KUKA KRL program: EPS_2_25694_BR02_A_20251117072400.src

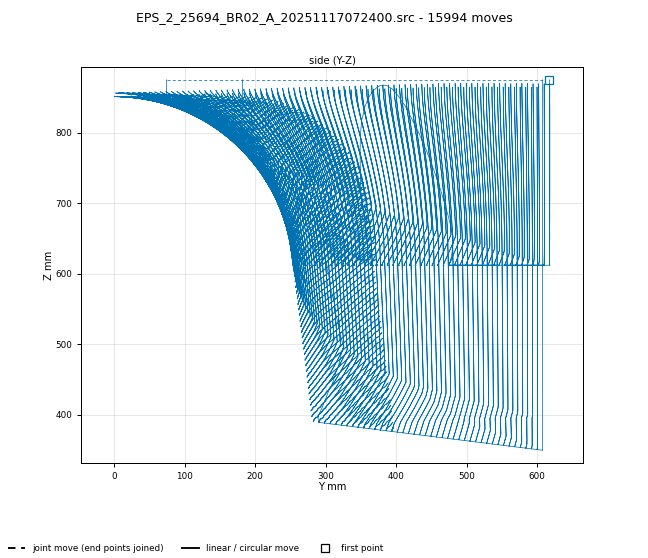
[picture p0: tool path of EPS_2_25694_BR02_A_20251117072400.src, 15994 of 15996 moves have a stored position in this frame; points joined in program order, loops and branches not executed]
&ACCESS RVP
&REL 4
&COMMENT QRS 19112012
&PARAM EDITMASK = *
DEF PART()
EXT BAS (BAS_COMMAND :IN,REAL :IN )
INT I
BAS (#INITMOV,0 )

;KUKA QRS Post kuka4.cps  Date:22-06-2017 !

File_ID=2912

QRS_PRE_INIT()

;Init var - Until changes are made in qrs_pre_init
Outlet_Square_prg=0
Inlet_1_Square_prg=0
Inlet_2_Square_prg=0
Inlet_3_Square_prg=0
Inlet_4_Square_prg=0
Inlet_5_Square_prg=0

Outlet_1={X 0.000, Y 466.000, Z 636.500, B 0.000, E1 0.000 }
Inlet_1={X 0.000, Y 492.670, Z 611.500, B 0.000, E1 180.000 }
Outlet_1_type=457
Inlet_1_type=0
;QRS#1=Sidecore dimensions
;QRS#2=450-18" Concrete
;QRS#3=DeadEnd 457
;QRS#4=
;QRS#5=
;QRS#6=
;QRS#7=
;QRS#8=
;QRS#9=28A PSX-2
;QRS#10=

;QRS#11=
;QRS#12=
;QRS#13=
;QRS#14=
;QRS#15=
;QRS#16=1220x127x1219 4'
;QRS#17=EPS Height
;QRS#18=865
;QRS#19=*
;QRS#20= UPDATED VERSION 22-06-2017
;QRS#21=*
Outlet_Square=0250
Inlet_1_Square=00
Inlet_2_Square=0
Inlet_3_Square=0
Inlet_4_Square=0
Inlet_5_Square=0
Mill_Square=1
Outlet_Square_Prg=274
Inlet_1_Square_prg=0

QRS_INIT()

$ADVANCE=5

; T1
PTP {E1 171.224,E2 171.224}
PTP {X 0,Y 617.539,A -85,B 0,C 180,E1 171.224,E2 171.224,E3 0,E4 0,E5 0,E6 0}
QRS_SPEED_INIT()
LIN {X 0,Y 617.539,Z 875,A -85,B 0,C 180,E1 171.224,E2 171.224,E3 0,E4 0,E5 0,E6 0} C_VEL
LIN {X 0,Y 617.539,Z 613.91,A -85,B 0,C 180,E1 171.224,E2 171.224} C_VEL
LIN {X 0,Y 617.52,Z 611.91,A -85,B 0,C 180,E1 171.41,E2 171.41} C_VEL
LIN {X 0,Y 618.01,Z 611.91,A -85,B 0,C 180,E1 174.219,E2 174.219} C_VEL
LIN {X 0,Y 618.036,Z 611.91,A -85,B 0,C 180,E1 178.849,E2 178.849} C_VEL
LIN {X 0,Y 617.996,Z 611.91,A -85,B 0,C 180,E1 183.472,E2 183.472} C_VEL
LIN {X 0,Y 617.993,Z 611.91,A -85,B 0,C 180,E1 188.118,E2 188.118} C_VEL
LIN {X 0,Y 617.979,Z 611.91,A -85,B 0,C 180,E1 192.819,E2 192.819} C_VEL
LIN {X 0,Y 617.92,Z 611.91,A -85,B 0,C 180,E1 197.611,E2 197.611} C_VEL
LIN {X 0,Y 617.739,Z 611.91,A -85,B 0,C 180,E1 198.543,E2 198.543} C_VEL
LIN {X 0,Y 617.926,Z 611.91,A -85,B 0,C 180,E1 202.533,E2 202.533} C_VEL
LIN {X 0,Y 617.417,Z 611.91,A -85,B 0,C 180,E1 205.081,E2 205.081} C_VEL
LIN {X 0,Y 617.847,Z 611.91,A -85,B 0,C 180,E1 207.641,E2 207.641} C_VEL
LIN {X 0,Y 617.342,Z 611.91,A -85,B 0,C 180,E1 210.31,E2 210.31} C_VEL
LIN {X 0,Y 617.812,Z 611.91,A -85,B 0,C 180,E1 213,E2 213} C_VEL
LIN {X 0,Y 617.679,Z 611.91,A -85,B 0,C 180,E1 214.194,E2 214.194} C_VEL
LIN {X 0,Y 617.782,Z 611.91,A -85,B 0,C 180,E1 218.707,E2 218.707} C_VEL
LIN {X 0,Y 617.421,Z 611.91,A -85,B 0,C 180,E1 221.764,E2 221.764} C_VEL
LIN {X 0,Y 617.823,Z 611.91,A -85,B 0,C 180,E1 224.908,E2 224.908} C_VEL
LIN {X 0,Y 617.772,Z 611.91,A -85,B 0,C 180,E1 228.277,E2 228.277} C_VEL
LIN {X 0,Y 617.551,Z 611.91,A -85,B 0,C 180,E1 231.279,E2 231.279} C_VEL
LIN {X 0,Y 617.574,Z 611.91,A -85,B 0,C 180,E1 231.903,E2 231.903} C_VEL
LIN {X 0,Y 617.811,Z 611.91,A -85,B 0,C 180,E1 234.203,E2 234.203} C_VEL
LIN {X 0,Y 617.347,Z 611.91,A -85,B 0,C 180,E1 236.976,E2 236.976} C_VEL
LIN {X 0,Y 617.893,Z 611.91,A -85,B 0,C 180,E1 239.723,E2 239.723} C_VEL
LIN {X 0,Y 618.039,Z 611.91,A -85,B 0,C 180,E1 244.95,E2 244.95} C_VEL
LIN {X 0,Y 617.661,Z 611.91,A -85,B 0,C 180,E1 245.064,E2 245.064} C_VEL
LIN {X 0,Y 617.895,Z 648.089,A -85,B 0,C 180,E1 245.541,E2 245.541} C_VEL
LIN {X 0,Y 617.86,Z 657.573,A -85,B 0,C 180,E1 245.694,E2 245.694} C_VEL
LIN {X 0,Y 617.789,Z 666.269,A -85,B 0,C 180,E1 245.863,E2 245.863} C_VEL
LIN {X 0,Y 617.896,Z 680.361,A -85,B 0,C 180,E1 246.223,E2 246.223} C_VEL
LIN {X 0,Y 617.817,Z 691.301,A -85,B 0,C 180,E1 246.552,E2 246.552} C_VEL
LIN {X 0,Y 617.928,Z 701.625,A -85,B 0,C 180,E1 246.918,E2 246.918} C_VEL
LIN {X 0,Y 617.942,Z 713.385,A -85,B 0,C 180,E1 247.393,E2 247.393} C_VEL
LIN {X 0,Y 617.876,Z 723.675,A -85,B 0,C 180,E1 247.859,E2 247.859} C_VEL
LIN {X 0,Y 617.946,Z 734.343,A -85,B 0,C 180,E1 248.407,E2 248.407} C_VEL
LIN {X 0,Y 617.967,Z 745.217,A -85,B 0,C 180,E1 249.027,E2 249.027} C_VEL
LIN {X 0,Y 617.938,Z 755.026,A -85,B 0,C 180,E1 249.644,E2 249.644} C_VEL
LIN {X 0,Y 617.951,Z 764.54,A -85,B 0,C 180,E1 250.302,E2 250.302} C_VEL
LIN {X 0,Y 617.956,Z 773.748,A -85,B 0,C 180,E1 251.001,E2 251.001} C_VEL
LIN {X 0,Y 617.967,Z 782.099,A -85,B 0,C 180,E1 251.691,E2 251.691} C_VEL
LIN {X 0,Y 617.941,Z 791.033,A -85,B 0,C 180,E1 252.497,E2 252.497} C_VEL
LIN {X 0,Y 617.896,Z 798.436,A -85,B 0,C 180,E1 253.222,E2 253.222} C_VEL
LIN {X 0,Y 617.951,Z 806.146,A -85,B 0,C 180,E1 254.049,E2 254.049} C_VEL
LIN {X 0,Y 617.974,Z 812.663,A -85,B 0,C 180,E1 254.803,E2 254.803} C_VEL
LIN {X 0,Y 617.884,Z 819.776,A -85,B 0,C 180,E1 255.697,E2 255.697} C_VEL
LIN {X 0,Y 617.866,Z 826.241,A -85,B 0,C 180,E1 256.589,E2 256.589} C_VEL
LIN {X 0,Y 617.965,Z 832.102,A -85,B 0,C 180,E1 257.481,E2 257.481} C_VEL
LIN {X 0,Y 617.877,Z 837.463,A -85,B 0,C 180,E1 258.365,E2 258.365} C_VEL
LIN {X 0,Y 617.831,Z 843.766,A -85,B 0,C 180,E1 259.542,E2 259.542} C_VEL
LIN {X 0,Y 617.913,Z 847.34,A -85,B 0,C 180,E1 260.283,E2 260.283} C_VEL
LIN {X 0,Y 617.929,Z 852.374,A -85,B 0,C 180,E1 261.453,E2 261.453} C_VEL
LIN {X 0,Y 617.831,Z 855.756,A -85,B 0,C 180,E1 262.35,E2 262.35} C_VEL
LIN {X 0,Y 617.936,Z 860.15,A -85,B 0,C 180,E1 263.748,E2 263.748} C_VEL
LIN {X 0,Y 617.913,Z 862.617,A -85,B 0,C 180,E1 264.677,E2 264.677} C_VEL
LIN {X 0,Y 617.775,Z 865.488,A -85,B 0,C 180,E1 266.068,E2 266.068} C_VEL
LIN {X 0,Y 617.811,Z 866.258,A -85,B 0,C 180,E1 266.531,E2 266.531} C_VEL
LIN {X 0,Y 617.948,Z 867.966,A -85,B 0,C 180,E1 267.92,E2 267.92} C_VEL
LIN {X 0,Y 617.798,Z 868.661,A -85,B 0,C 180,E1 268.844,E2 268.844} C_VEL
LIN {X 0,Y 617.834,Z 868.908,A -85,B 0,C 180,E1 270.231,E2 270.231} C_VEL
LIN {X 0,Y 617.983,Z 868.61,A -85,B 0,C 180,E1 271.155,E2 271.155} C_VEL
LIN {X 0,Y 617.813,Z 867.476,A -85,B 0,C 180,E1 272.543,E2 272.543} C_VEL
LIN {X 0,Y 617.843,Z 866.25,A -85,B 0,C 180,E1 273.469,E2 273.469} C_VEL
LIN {X 0,Y 617.982,Z 864.618,A -85,B 0,C 180,E1 274.395,E2 274.395} C_VEL
LIN {X 0,Y 617.84,Z 862.636,A -85,B 0,C 180,E1 275.323,E2 275.323} C_VEL
LIN {X 0,Y 617.779,Z 860.19,A -85,B 0,C 180,E1 276.253,E2 276.253} C_VEL
LIN {X 0,Y 617.946,Z 855.728,A -85,B 0,C 180,E1 277.648,E2 277.648} C_VEL
LIN {X 0,Y 617.875,Z 851.36,A -85,B 0,C 180,E1 278.793,E2 278.793} C_VEL
LIN {X 0,Y 617.822,Z 847.625,A -85,B 0,C 180,E1 279.664,E2 279.664} C_VEL
LIN {X 0,Y 617.935,Z 842.258,A -85,B 0,C 180,E1 280.75,E2 280.75} C_VEL
LIN {X 0,Y 617.942,Z 837.449,A -85,B 0,C 180,E1 281.634,E2 281.634} C_VEL
LIN {X 0,Y 617.865,Z 830.198,A -85,B 0,C 180,E1 282.818,E2 282.818} C_VEL
LIN {X 0,Y 617.941,Z 824.137,A -85,B 0,C 180,E1 283.706,E2 283.706} C_VEL
LIN {X 0,Y 617.959,Z 817.47,A -85,B 0,C 180,E1 284.6,E2 284.6} C_VEL
LIN {X 0,Y 617.884,Z 809.516,A -85,B 0,C 180,E1 285.57,E2 285.57} C_VEL
LIN {X 0,Y 617.919,Z 802.465,A -85,B 0,C 180,E1 286.355,E2 286.355} C_VEL
LIN {X 0,Y 617.972,Z 794.297,A -85,B 0,C 180,E1 287.187,E2 287.187} C_VEL
LIN {X 0,Y 617.934,Z 787.157,A -85,B 0,C 180,E1 287.863,E2 287.863} C_VEL
LIN {X 0,Y 617.923,Z 778.285,A -85,B 0,C 180,E1 288.631,E2 288.631} C_VEL
LIN {X 0,Y 617.943,Z 769.373,A -85,B 0,C 180,E1 289.338,E2 289.338} C_VEL
LIN {X 0,Y 617.96,Z 760.865,A -85,B 0,C 180,E1 289.959,E2 289.959} C_VEL
LIN {X 0,Y 617.96,Z 751.47,A -85,B 0,C 180,E1 290.587,E2 290.587} C_VEL
LIN {X 0,Y 617.918,Z 741.279,A -85,B 0,C 180,E1 291.207,E2 291.207} C_VEL
LIN {X 0,Y 617.943,Z 731.417,A -85,B 0,C 180,E1 291.749,E2 291.749} C_VEL
LIN {X 0,Y 617.958,Z 720.361,A -85,B 0,C 180,E1 292.294,E2 292.294} C_VEL
LIN {X 0,Y 617.921,Z 709.648,A -85,B 0,C 180,E1 292.766,E2 292.766} C_VEL
LIN {X 0,Y 617.818,Z 698.36,A -85,B 0,C 180,E1 293.205,E2 293.205} C_VEL
LIN {X 0,Y 617.93,Z 686.204,A -85,B 0,C 180,E1 293.604,E2 293.604} C_VEL
LIN {X 0,Y 617.911,Z 675,A -85,B 0,C 180,E1 293.92,E2 293.92} C_VEL
LIN {X 0,Y 617.75,Z 663.936,A -85,B 0,C 180,E1 294.186,E2 294.186} C_VEL
LIN {X 0,Y 617.899,Z 651.747,A -85,B 0,C 180,E1 294.405,E2 294.405} C_VEL
LIN {X 0,Y 617.853,Z 635.322,A -85,B 0,C 180,E1 294.632,E2 294.632} C_VEL
LIN {X 0,Y 617.679,Z 611.91,A -85,B 0,C 180,E1 294.936,E2 294.936} C_VEL
LIN {X 0,Y 618.055,Z 611.91,A -85,B 0,C 180,E1 295.049,E2 295.049} C_VEL
LIN {X 0,Y 617.893,Z 611.91,A -85,B 0,C 180,E1 300.277,E2 300.277} C_VEL
LIN {X 0,Y 617.347,Z 611.91,A -85,B 0,C 180,E1 303.024,E2 303.024} C_VEL
LIN {X 0,Y 617.811,Z 611.91,A -85,B 0,C 180,E1 305.797,E2 305.797} C_VEL
LIN {X 0,Y 617.546,Z 611.91,A -85,B 0,C 180,E1 308.721,E2 308.721} C_VEL
LIN {X 0,Y 617.75,Z 611.91,A -85,B 0,C 180,E1 311.733,E2 311.733} C_VEL
LIN {X 0,Y 617.804,Z 611.91,A -85,B 0,C 180,E1 315.09,E2 315.09} C_VEL
LIN {X 0,Y 617.418,Z 611.91,A -85,B 0,C 180,E1 318.31,E2 318.31} C_VEL
LIN {X 0,Y 617.776,Z 611.91,A -85,B 0,C 180,E1 321.292,E2 321.292} C_VEL
LIN {X 0,Y 617.679,Z 611.91,A -85,B 0,C 180,E1 325.806,E2 325.806} C_VEL
LIN {X 0,Y 617.847,Z 611.91,A -85,B 0,C 180,E1 327.002,E2 327.002} C_VEL
LIN {X 0,Y 617.633,Z 611.91,A -85,B 0,C 180,E1 330.175,E2 330.175} C_VEL
LIN {X 0,Y 617.65,Z 611.91,A -85,B 0,C 180,E1 332.349,E2 332.349} C_VEL
LIN {X 0,Y 617.509,Z 611.91,A -85,B 0,C 180,E1 335.241,E2 335.241} C_VEL
LIN {X 0,Y 617.715,Z 611.91,A -85,B 0,C 180,E1 337.459,E2 337.459} C_VEL
LIN {X 0,Y 617.711,Z 611.91,A -85,B 0,C 180,E1 341.465,E2 341.465} C_VEL
LIN {X 0,Y 617.915,Z 611.91,A -85,B 0,C 180,E1 342.389,E2 342.389} C_VEL
LIN {X 0,Y 617.972,Z 611.91,A -85,B 0,C 180,E1 347.181,E2 347.181} C_VEL
LIN {X 0,Y 617.987,Z 611.91,A -85,B 0,C 180,E1 351.882,E2 351.882} C_VEL
LIN {X 0,Y 617.986,Z 611.91,A -85,B 0,C 180,E1 356.528,E2 356.528} C_VEL
LIN {X 0,Y 618.036,Z 611.91,A -85,B 0,C 180,E1 361.151,E2 361.151} C_VEL
LIN {X 0,Y 618.009,Z 611.91,A -85,B 0,C 180,E1 365.781,E2 365.781} C_VEL
LIN {X 0,Y 617.945,Z 611.91,A -85,B 0,C 180,E1 370.451,E2 370.451} C_VEL
LIN {X 0,Y 617.949,Z 611.91,A -85,B 0,C 180,E1 375.192,E2 375.192} C_VEL
LIN {X 0,Y 617.917,Z 611.91,A -85,B 0,C 180,E1 380.044,E2 380.044} C_VEL
LIN {X 0,Y 617.427,Z 611.91,A -85,B 0,C 180,E1 382.542,E2 382.542} C_VEL
LIN {X 0,Y 617.87,Z 611.91,A -85,B 0,C 180,E1 385.051,E2 385.051} C_VEL
LIN {X 0,Y 617.368,Z 611.91,A -85,B 0,C 180,E1 387.654,E2 387.654} C_VEL
LIN {X 0,Y 617.822,Z 611.91,A -85,B 0,C 180,E1 390.274,E2 390.274} C_VEL
LIN {X 0,Y 617.306,Z 611.91,A -85,B 0,C 180,E1 393.02,E2 393.02} C_VEL
LIN {X 0,Y 617.795,Z 611.91,A -85,B 0,C 180,E1 395.791,E2 395.791} C_VEL
LIN {X 0,Y 617.874,Z 611.91,A -85,B 0,C 180,E1 398.689,E2 398.689} C_VEL
LIN {X 0,Y 617.401,Z 611.91,A -85,B 0,C 180,E1 401.754,E2 401.754} C_VEL
LIN {X 0,Y 617.853,Z 611.91,A -85,B 0,C 180,E1 404.893,E2 404.893} C_VEL
LIN {X 0,Y 617.725,Z 611.91,A -85,B 0,C 180,E1 408.269,E2 408.269} C_VEL
LIN {X 0,Y 617.496,Z 611.91,A -85,B 0,C 180,E1 411.275,E2 411.275} C_VEL
LIN {X 0,Y 617.519,Z 611.91,A -85,B 0,C 180,E1 411.895,E2 411.895} C_VEL
LIN {X 0,Y 617.754,Z 611.91,A -85,B 0,C 180,E1 414.199,E2 414.199} C_VEL
LIN {X 0,Y 617.28,Z 611.91,A -85,B 0,C 180,E1 416.972,E2 416.972} C_VEL
LIN {X 0,Y 617.815,Z 611.91,A -85,B 0,C 180,E1 419.719,E2 419.719} C_VEL
LIN {X 0,Y 617.39,Z 611.91,A -85,B 0,C 180,E1 422.34,E2 422.34} C_VEL
LIN {X 0,Y 617.915,Z 611.91,A -85,B 0,C 180,E1 424.945,E2 424.945} C_VEL
LIN {X 0,Y 617.43,Z 611.91,A -85,B 0,C 180,E1 427.452,E2 427.452} C_VEL
LIN {X 0,Y 617.885,Z 611.91,A -85,B 0,C 180,E1 429.95,E2 429.95} C_VEL
LIN {X 0,Y 617.964,Z 611.91,A -85,B 0,C 180,E1 434.803,E2 434.803} C_VEL
LIN {X 0,Y 617.954,Z 611.91,A -85,B 0,C 180,E1 439.544,E2 439.544} C_VEL
LIN {X 0,Y 617.973,Z 611.91,A -85,B 0,C 180,E1 444.213,E2 444.213} C_VEL
LIN {X 0,Y 618.038,Z 611.91,A -85,B 0,C 180,E1 448.845,E2 448.845} C_VEL
LIN {X 0,Y 618.005,Z 611.91,A -85,B 0,C 180,E1 453.468,E2 453.468} C_VEL
LIN {X 0,Y 617.96,Z 611.91,A -85,B 0,C 180,E1 458.115,E2 458.115} C_VEL
LIN {X 0,Y 617.98,Z 611.91,A -85,B 0,C 180,E1 462.815,E2 462.815} C_VEL
LIN {X 0,Y 617.923,Z 611.91,A -85,B 0,C 180,E1 467.607,E2 467.607} C_VEL
LIN {X 0,Y 617.736,Z 611.91,A -85,B 0,C 180,E1 468.563,E2 468.563} C_VEL
LIN {X 0,Y 617.884,Z 611.91,A -85,B 0,C 180,E1 472.531,E2 472.531} C_VEL
LIN {X 0,Y 617.394,Z 611.91,A -85,B 0,C 180,E1 475.078,E2 475.078} C_VEL
LIN {X 0,Y 617.847,Z 611.91,A -85,B 0,C 180,E1 477.638,E2 477.638} C_VEL
LIN {X 0,Y 617.404,Z 611.91,A -85,B 0,C 180,E1 480.303,E2 480.303} C_VEL
LIN {X 0,Y 617.946,Z 611.91,A -85,B 0,C 180,E1 482.988,E2 482.988} C_VEL
LIN {X 0,Y 617.681,Z 611.91,A -85,B 0,C 180,E1 485.806,E2 485.806} C_VEL
LIN {X 0,Y 617.68,Z 611.91,A -85,B 0,C 180,E1 488.124,E2 488.124} C_VEL
LIN {X 0,Y 617.747,Z 611.91,A -85,B 0,C 180,E1 491.734,E2 491.734} C_VEL
LIN {X 0,Y 617.388,Z 611.91,A -85,B 0,C 180,E1 495.064,E2 495.064} C_VEL
LIN {X 0,Y 617.754,Z 611.91,A -85,B 0,C 180,E1 498.275,E2 498.275} C_VEL
LIN {X 0,Y 617.342,Z 611.91,A -85,B 0,C 180,E1 501.926,E2 501.926} C_VEL
LIN {X 0,Y 617.807,Z 611.91,A -85,B 0,C 180,E1 504.21,E2 504.21} C_VEL
LIN {X 0,Y 617.305,Z 611.91,A -85,B 0,C 180,E1 506.98,E2 506.98} C_VEL
LIN {X 0,Y 617.828,Z 611.91,A -85,B 0,C 180,E1 509.726,E2 509.726} C_VEL
LIN {X 0,Y 617.374,Z 611.91,A -85,B 0,C 180,E1 512.346,E2 512.346} C_VEL
LIN {X 0,Y 617.876,Z 611.91,A -85,B 0,C 180,E1 514.949,E2 514.949} C_VEL
LIN {X 0,Y 617.433,Z 611.91,A -85,B 0,C 180,E1 517.458,E2 517.458} C_VEL
LIN {X 0,Y 617.944,Z 611.91,A -85,B 0,C 180,E1 519.957,E2 519.957} C_VEL
LIN {X 0,Y 618.009,Z 611.91,A -85,B 0,C 180,E1 523.637,E2 523.637} C_VEL
LIN {X 0,Y 617.952,Z 611.91,A -85,B 0,C 180,E1 529.549,E2 529.549} C_VEL
LIN {X 0,Y 617.52,Z 611.91,A -85,B 0,C 180,E1 531.41,E2 531.41} C_VEL
LIN {X 0,Y 613.85,Z 611.91,A -85,B 0,C 180,E1 533.002,E2 533.002} C_VEL
LIN {X 0,Y 609.957,Z 611.91,A -85,B 0,C 180,E1 534.613,E2 534.613} C_VEL
LIN {X 0,Y 609.775,Z 611.91,A -85,B 0,C 180,E1 539.997,E2 539.997} C_VEL
LIN {X 0,Y 609.833,Z 611.91,A -85,B 0,C 180,E1 544.269,E2 544.269} C_VEL
LIN {X 0,Y 609.922,Z 611.91,A -85,B 0,C 180,E1 548.563,E2 548.563} C_VEL
LIN {X 0,Y 610.05,Z 611.91,A -85,B 0,C 180,E1 552.904,E2 552.904} C_VEL
LIN {X 0,Y 609.778,Z 611.91,A -85,B 0,C 180,E1 558.828,E2 558.828} C_VEL
LIN {X 0,Y 609.722,Z 611.91,A -85,B 0,C 180,E1 563.406,E2 563.406} C_VEL
LIN {X 0,Y 609.766,Z 611.91,A -85,B 0,C 180,E1 568.145,E2 568.145} C_VEL
LIN {X 0,Y 609.919,Z 611.91,A -85,B 0,C 180,E1 573.097,E2 573.097} C_VEL
LIN {X 0,Y 609.599,Z 611.91,A -85,B 0,C 180,E1 579.651,E2 579.651} C_VEL
LIN {X 0,Y 609.699,Z 611.91,A -85,B 0,C 180,E1 585.947,E2 585.947} C_VEL
LIN {X 0,Y 609.553,Z 611.91,A -85,B 0,C 180,E1 590.347,E2 590.347} C_VEL
LIN {X 0,Y 609.601,Z 611.91,A -85,B 0,C 180,E1 595.163,E2 595.163} C_VEL
LIN {X 0,Y 609.769,Z 611.91,A -85,B 0,C 180,E1 600.339,E2 600.339} C_VEL
LIN {X 0,Y 610.013,Z 611.91,A -85,B 0,C 180,E1 604.709,E2 604.709} C_VEL
LIN {X 0,Y 610.606,Z 670.171,A -85,B 0,C 180,E1 605.655,E2 605.655} C_VEL
LIN {X 0,Y 610.583,Z 705.337,A -85,B 0,C 180,E1 606.772,E2 606.772} C_VEL
LIN {X 0,Y 610.488,Z 739.951,A -85,B 0,C 180,E1 608.447,E2 608.447} C_VEL
LIN {X 0,Y 610.346,Z 772.524,A -85,B 0,C 180,E1 610.652,E2 610.652} C_VEL
LIN {X 0,Y 610.183,Z 800.75,A -85,B 0,C 180,E1 613.235,E2 613.235} C_VEL
LIN {X 0,Y 610.082,Z 824.976,A -85,B 0,C 180,E1 616.18,E2 616.18} C_VEL
LIN {X 0,Y 610.02,Z 843.72,A -85,B 0,C 180,E1 619.272,E2 619.272} C_VEL
LIN {X 0,Y 610.037,Z 856.977,A -85,B 0,C 180,E1 622.369,E2 622.369} C_VEL
LIN {X 0,Y 609.982,Z 865.971,A -85,B 0,C 180,E1 625.73,E2 625.73} C_VEL
LIN {X 0,Y 610.021,Z 869.507,A -85,B 0,C 180,E1 628.578,E2 628.578} C_VEL
LIN {X 0,Y 610.115,Z 869.507,A -85,B 0,C 180,E1 631.422,E2 631.422} C_VEL
LIN {X 0,Y 610.052,Z 864.451,A -85,B 0,C 180,E1 634.983,E2 634.983} C_VEL
LIN {X 0,Y 610.081,Z 853.497,A -85,B 0,C 180,E1 638.563,E2 638.563} C_VEL
LIN {X 0,Y 610.103,Z 836.711,A -85,B 0,C 180,E1 641.996,E2 641.996} C_VEL
LIN {X 0,Y 610.163,Z 815.396,A -85,B 0,C 180,E1 645.086,E2 645.086} C_VEL
LIN {X 0,Y 610.254,Z 788.575,A -85,B 0,C 180,E1 647.974,E2 647.974} C_VEL
LIN {X 0,Y 610.403,Z 757.994,A -85,B 0,C 180,E1 650.414,E2 650.414} C_VEL
LIN {X 0,Y 610.533,Z 725.726,A -85,B 0,C 180,E1 652.317,E2 652.317} C_VEL
LIN {X 0,Y 610.661,Z 689.318,A -85,B 0,C 180,E1 653.808,E2 653.808} C_VEL
LIN {X 0,Y 610.724,Z 653.487,A -85,B 0,C 180,E1 654.684,E2 654.684} C_VEL
LIN {X 0,Y 610.027,Z 611.91,A -85,B 0,C 180,E1 655.29,E2 655.29} C_VEL
LIN {X 0,Y 609.599,Z 611.91,A -85,B 0,C 180,E1 661.438,E2 661.438} C_VEL
LIN {X 0,Y 609.712,Z 611.91,A -85,B 0,C 180,E1 666.582,E2 666.582} C_VEL
LIN {X 0,Y 609.752,Z 611.91,A -85,B 0,C 180,E1 672.1,E2 672.1} C_VEL
LIN {X 0,Y 609.475,Z 611.91,A -85,B 0,C 180,E1 677.882,E2 677.882} C_VEL
LIN {X 0,Y 609.46,Z 611.91,A -85,B 0,C 180,E1 682.652,E2 682.652} C_VEL
LIN {X 0,Y 609.795,Z 611.91,A -85,B 0,C 180,E1 687.584,E2 687.584} C_VEL
LIN {X 0,Y 609.685,Z 611.91,A -85,B 0,C 180,E1 691.851,E2 691.851} C_VEL
LIN {X 0,Y 609.651,Z 611.91,A -85,B 0,C 180,E1 696.764,E2 696.764} C_VEL
LIN {X 0,Y 609.914,Z 611.91,A -85,B 0,C 180,E1 702.673,E2 702.673} C_VEL
LIN {X 0,Y 610.028,Z 611.91,A -85,B 0,C 180,E1 707.096,E2 707.096} C_VEL
LIN {X 0,Y 609.768,Z 611.91,A -85,B 0,C 180,E1 712.871,E2 712.871} C_VEL
LIN {X 0,Y 609.867,Z 611.91,A -85,B 0,C 180,E1 717.157,E2 717.157} C_VEL
LIN {X 0,Y 610.021,Z 611.91,A -85,B 0,C 180,E1 721.425,E2 721.425} C_VEL
LIN {X 0,Y 609.773,Z 611.91,A -85,B 0,C 180,E1 726.69,E2 726.69} C_VEL
LIN {X 0,Y 609.707,Z 611.91,A -85,B 0,C 180,E1 731.461,E2 731.461} C_VEL
LIN {X 0,Y 609.796,Z 611.91,A -85,B 0,C 180,E1 735.852,E2 735.852} C_VEL
LIN {X 0,Y 609.897,Z 611.91,A -85,B 0,C 180,E1 740.339,E2 740.339} C_VEL
LIN {X 0,Y 609.95,Z 611.91,A -85,B 0,C 180,E1 744.962,E2 744.962} C_VEL
LIN {X 0,Y 609.743,Z 611.91,A -85,B 0,C 180,E1 749.778,E2 749.778} C_VEL
LIN {X 0,Y 609.764,Z 611.91,A -85,B 0,C 180,E1 756.58,E2 756.58} C_VEL
LIN {X 0,Y 609.515,Z 611.91,A -85,B 0,C 180,E1 761.823,E2 761.823} C_VEL
LIN {X 0,Y 609.667,Z 611.91,A -85,B 0,C 180,E1 766.071,E2 766.071} C_VEL
LIN {X 0,Y 609.487,Z 611.91,A -85,B 0,C 180,E1 770.363,E2 770.363} C_VEL
LIN {X 0,Y 609.548,Z 611.91,A -85,B 0,C 180,E1 775.159,E2 775.159} C_VEL
LIN {X 0,Y 609.698,Z 611.91,A -85,B 0,C 180,E1 780.361,E2 780.361} C_VEL
LIN {X 0,Y 609.988,Z 611.91,A -85,B 0,C 180,E1 785.042,E2 785.042} C_VEL
LIN {X 0,Y 609.714,Z 611.91,A -85,B 0,C 180,E1 790.67,E2 790.67} C_VEL
LIN {X 0,Y 609.77,Z 611.91,A -85,B 0,C 180,E1 795.623,E2 795.623} C_VEL
LIN {X 0,Y 609.888,Z 611.91,A -85,B 0,C 180,E1 799.993,E2 799.993} C_VEL
LIN {X 0,Y 610.054,Z 611.91,A -85,B 0,C 180,E1 804.303,E2 804.303} C_VEL
LIN {X 0,Y 609.757,Z 611.91,A -85,B 0,C 180,E1 810,E2 810} C_VEL
LIN {X 0,Y 609.805,Z 611.91,A -85,B 0,C 180,E1 814.272,E2 814.272} C_VEL
LIN {X 0,Y 609.899,Z 611.91,A -85,B 0,C 180,E1 818.566,E2 818.566} C_VEL
LIN {X 0,Y 610.032,Z 611.91,A -85,B 0,C 180,E1 822.907,E2 822.907} C_VEL
LIN {X 0,Y 609.75,Z 611.91,A -85,B 0,C 180,E1 828.832,E2 828.832} C_VEL
LIN {X 0,Y 609.675,Z 611.91,A -85,B 0,C 180,E1 833.412,E2 833.412} C_VEL
LIN {X 0,Y 609.767,Z 611.91,A -85,B 0,C 180,E1 838.149,E2 838.149} C_VEL
LIN {X 0,Y 610.006,Z 611.91,A -85,B 0,C 180,E1 843.096,E2 843.096} C_VEL
LIN {X 0,Y 609.719,Z 611.91,A -85,B 0,C 180,E1 848.375,E2 848.375} C_VEL
LIN {X 0,Y 609.729,Z 611.91,A -85,B 0,C 180,E1 852.102,E2 852.102} C_VEL
LIN {X 0,Y 609.824,Z 611.91,A -85,B 0,C 180,E1 858.145,E2 858.145} C_VEL
LIN {X 0,Y 609.615,Z 611.91,A -85,B 0,C 180,E1 865.044,E2 865.044} C_VEL
LIN {X 0,Y 609.73,Z 611.91,A -85,B 0,C 180,E1 870.355,E2 870.355} C_VEL
LIN {X 0,Y 609.966,Z 611.91,A -85,B 0,C 180,E1 875.039,E2 875.039} C_VEL
LIN {X 0,Y 609.814,Z 611.91,A -85,B 0,C 180,E1 881.168,E2 881.168} C_VEL
LIN {X 0,Y 609.34,Z 611.91,A -85,B 0,C 180,E1 885.708,E2 885.708} C_VEL
LIN {X 0,Y 609.896,Z 611.91,A -85,B 0,C 180,E1 889.991,E2 889.991} C_VEL
LIN {X 0,Y 609.957,Z 611.91,A -85,B 0,C 180,E1 894.613,E2 894.613} C_VEL
LIN {X 0,Y 605.701,Z 611.91,A -85,B 0,C 180,E1 896.209,E2 896.209} C_VEL
LIN {X 0,Y 601.909,Z 611.91,A -85,B 0,C 180,E1 897.827,E2 897.827} C_VEL
LIN {X 0,Y 601.975,Z 611.91,A -85,B 0,C 180,E1 902.881,E2 902.881} C_VEL
LIN {X 0,Y 601.98,Z 611.91,A -85,B 0,C 180,E1 908.677,E2 908.677} C_VEL
LIN {X 0,Y 602.073,Z 611.91,A -85,B 0,C 180,E1 913.078,E2 913.078} C_VEL
LIN {X 0,Y 601.826,Z 611.91,A -85,B 0,C 180,E1 919.086,E2 919.086} C_VEL
LIN {X 0,Y 601.744,Z 611.91,A -85,B 0,C 180,E1 923.736,E2 923.736} C_VEL
LIN {X 0,Y 601.753,Z 611.91,A -85,B 0,C 180,E1 928.554,E2 928.554} C_VEL
LIN {X 0,Y 601.8,Z 611.91,A -85,B 0,C 180,E1 933.877,E2 933.877} C_VEL
LIN {X 0,Y 601.753,Z 611.91,A -85,B 0,C 180,E1 938.972,E2 938.972} C_VEL
LIN {X 0,Y 601.696,Z 611.91,A -85,B 0,C 180,E1 945.205,E2 945.205} C_VEL
LIN {X 0,Y 601.698,Z 611.91,A -85,B 0,C 180,E1 951.018,E2 951.018} C_VEL
LIN {X 0,Y 601.55,Z 611.91,A -85,B 0,C 180,E1 956.151,E2 956.151} C_VEL
LIN {X 0,Y 601.605,Z 611.91,A -85,B 0,C 180,E1 961.434,E2 961.434} C_VEL
LIN {X 0,Y 601.954,Z 611.91,A -85,B 0,C 180,E1 964.333,E2 964.333} C_VEL
LIN {X 0,Y 603.403,Z 619.37,A -85,B 0,C 180,E1 964.531,E2 964.531} C_VEL
LIN {X 0,Y 603.397,Z 670.167,A -85,B 0,C 180,E1 965.345,E2 965.345} C_VEL
LIN {X 0,Y 603.257,Z 706.431,A -85,B 0,C 180,E1 966.518,E2 966.518} C_VEL
LIN {X 0,Y 603.016,Z 739.941,A -85,B 0,C 180,E1 968.166,E2 968.166} C_VEL
LIN {X 0,Y 602.747,Z 772.515,A -85,B 0,C 180,E1 970.398,E2 970.398} C_VEL
LIN {X 0,Y 602.437,Z 800.828,A -85,B 0,C 180,E1 973.02,E2 973.02} C_VEL
LIN {X 0,Y 602.281,Z 824.976,A -85,B 0,C 180,E1 975.998,E2 975.998} C_VEL
LIN {X 0,Y 602.155,Z 844.349,A -85,B 0,C 180,E1 979.261,E2 979.261} C_VEL
LIN {X 0,Y 602.141,Z 857.462,A -85,B 0,C 180,E1 982.414,E2 982.414} C_VEL
LIN {X 0,Y 602.103,Z 865.972,A -85,B 0,C 180,E1 985.674,E2 985.674} C_VEL
LIN {X 0,Y 602.12,Z 869.51,A -85,B 0,C 180,E1 988.559,E2 988.559} C_VEL
LIN {X 0,Y 602.21,Z 869.51,A -85,B 0,C 180,E1 991.441,E2 991.441} C_VEL
LIN {X 0,Y 602.161,Z 864.449,A -85,B 0,C 180,E1 995.049,E2 995.049} C_VEL
LIN {X 0,Y 602.186,Z 853.501,A -85,B 0,C 180,E1 998.677,E2 998.677} C_VEL
LIN {X 0,Y 602.249,Z 836.715,A -85,B 0,C 180,E1 1002.154,E2 1002.154} C_VEL
LIN {X 0,Y 602.401,Z 815.261,A -85,B 0,C 180,E1 1005.302,E2 1005.302} C_VEL
LIN {X 0,Y 602.599,Z 788.574,A -85,B 0,C 180,E1 1008.21,E2 1008.21} C_VEL
LIN {X 0,Y 602.867,Z 757.327,A -85,B 0,C 180,E1 1010.728,E2 1010.728} C_VEL
LIN {X 0,Y 603.163,Z 723.303,A -85,B 0,C 180,E1 1012.73,E2 1012.73} C_VEL
LIN {X 0,Y 603.401,Z 687.763,A -85,B 0,C 180,E1 1014.162,E2 1014.162} C_VEL
LIN {X 0,Y 603.552,Z 652.332,A -85,B 0,C 180,E1 1015.015,E2 1015.015} C_VEL
LIN {X 0,Y 602.951,Z 615.598,A -85,B 0,C 180,E1 1015.538,E2 1015.538} C_VEL
LIN {X 0,Y 601.944,Z 611.91,A -85,B 0,C 180,E1 1015.715,E2 1015.715} C_VEL
LIN {X 0,Y 601.631,Z 611.91,A -85,B 0,C 180,E1 1021.903,E2 1021.903} C_VEL
LIN {X 0,Y 601.717,Z 611.91,A -85,B 0,C 180,E1 1027.149,E2 1027.149} C_VEL
LIN {X 0,Y 601.726,Z 611.91,A -85,B 0,C 180,E1 1033.146,E2 1033.146} C_VEL
LIN {X 0,Y 601.534,Z 611.91,A -85,B 0,C 180,E1 1039.13,E2 1039.13} C_VEL
LIN {X 0,Y 601.462,Z 611.91,A -85,B 0,C 180,E1 1043.662,E2 1043.662} C_VEL
LIN {X 0,Y 601.791,Z 611.91,A -85,B 0,C 180,E1 1048.111,E2 1048.111} C_VEL
LIN {X 0,Y 601.648,Z 611.91,A -85,B 0,C 180,E1 1053.07,E2 1053.07} C_VEL
LIN {X 0,Y 601.63,Z 611.91,A -85,B 0,C 180,E1 1058.613,E2 1058.613} C_VEL
LIN {X 0,Y 601.925,Z 611.91,A -85,B 0,C 180,E1 1062.908,E2 1062.908} C_VEL
LIN {X 0,Y 601.811,Z 611.91,A -85,B 0,C 180,E1 1068.392,E2 1068.392} C_VEL
LIN {X 0,Y 601.867,Z 611.91,A -85,B 0,C 180,E1 1072.777,E2 1072.777} C_VEL
LIN {X 0,Y 601.971,Z 611.91,A -85,B 0,C 180,E1 1077.119,E2 1077.119} C_VEL
LIN {X 0,Y 602.11,Z 611.91,A -85,B 0,C 180,E1 1081.443,E2 1081.443} C_VEL
LIN {X 0,Y 602.178,Z 611.91,A -85,B 0,C 180,E1 1085.774,E2 1085.774} C_VEL
LIN {X 0,Y 601.796,Z 611.91,A -85,B 0,C 180,E1 1091.613,E2 1091.613} C_VEL
LIN {X 0,Y 601.829,Z 611.91,A -85,B 0,C 180,E1 1096.067,E2 1096.067} C_VEL
LIN {X 0,Y 601.727,Z 611.91,A -85,B 0,C 180,E1 1101.411,E2 1101.411} C_VEL
LIN {X 0,Y 601.939,Z 611.91,A -85,B 0,C 180,E1 1105.317,E2 1105.317} C_VEL
LIN {X 0,Y 601.637,Z 611.91,A -85,B 0,C 180,E1 1111.171,E2 1111.171} C_VEL
LIN {X 0,Y 601.849,Z 611.91,A -85,B 0,C 180,E1 1117.141,E2 1117.141} C_VEL
LIN {X 0,Y 601.582,Z 611.91,A -85,B 0,C 180,E1 1123.125,E2 1123.125} C_VEL
LIN {X 0,Y 601.752,Z 611.91,A -85,B 0,C 180,E1 1127.208,E2 1127.208} C_VEL
LIN {X 0,Y 601.722,Z 611.91,A -85,B 0,C 180,E1 1132.851,E2 1132.851} C_VEL
LIN {X 0,Y 601.625,Z 611.91,A -85,B 0,C 180,E1 1138.832,E2 1138.832} C_VEL
LIN {X 0,Y 602.032,Z 611.91,A -85,B 0,C 180,E1 1144.874,E2 1144.874} C_VEL
LIN {X 0,Y 601.768,Z 611.91,A -85,B 0,C 180,E1 1150.908,E2 1150.908} C_VEL
LIN {X 0,Y 601.906,Z 611.91,A -85,B 0,C 180,E1 1155.431,E2 1155.431} C_VEL
LIN {X 0,Y 601.955,Z 611.91,A -85,B 0,C 180,E1 1159.859,E2 1159.859} C_VEL
LIN {X 0,Y 602.143,Z 611.91,A -85,B 0,C 180,E1 1164.228,E2 1164.228} C_VEL
LIN {X 0,Y 601.857,Z 611.91,A -85,B 0,C 180,E1 1170,E2 1170} C_VEL
LIN {X 0,Y 601.901,Z 611.91,A -85,B 0,C 180,E1 1174.328,E2 1174.328} C_VEL
LIN {X 0,Y 601.958,Z 611.91,A -85,B 0,C 180,E1 1178.68,E2 1178.68} C_VEL
LIN {X 0,Y 602.054,Z 611.91,A -85,B 0,C 180,E1 1183.081,E2 1183.081} C_VEL
LIN {X 0,Y 601.801,Z 611.91,A -85,B 0,C 180,E1 1189.091,E2 1189.091} C_VEL
LIN {X 0,Y 601.701,Z 611.91,A -85,B 0,C 180,E1 1193.741,E2 1193.741} C_VEL
LIN {X 0,Y 601.768,Z 611.91,A -85,B 0,C 180,E1 1198.558,E2 1198.558} C_VEL
LIN {X 0,Y 601.91,Z 611.91,A -85,B 0,C 180,E1 1203.891,E2 1203.891} C_VEL
LIN {X 0,Y 601.716,Z 611.91,A -85,B 0,C 180,E1 1208.981,E2 1208.981} C_VEL
LIN {X 0,Y 601.564,Z 611.91,A -85,B 0,C 180,E1 1213.122,E2 1213.122} C_VEL
LIN {X 0,Y 601.603,Z 611.91,A -85,B 0,C 180,E1 1219.129,E2 1219.129} C_VEL
LIN {X 0,Y 601.683,Z 611.91,A -85,B 0,C 180,E1 1224.635,E2 1224.635} C_VEL
LIN {X 0,Y 601.748,Z 611.91,A -85,B 0,C 180,E1 1229.785,E2 1229.785} C_VEL
LIN {X 0,Y 602.017,Z 611.91,A -85,B 0,C 180,E1 1234.876,E2 1234.876} C_VEL
LIN {X 0,Y 601.942,Z 611.91,A -85,B 0,C 180,E1 1240.912,E2 1240.912} C_VEL
LIN {X 0,Y 601.513,Z 611.91,A -85,B 0,C 180,E1 1245.419,E2 1245.419} C_VEL
LIN {X 0,Y 601.949,Z 611.91,A -85,B 0,C 180,E1 1249.857,E2 1249.857} C_VEL
LIN {X 0,Y 602.037,Z 611.91,A -85,B 0,C 180,E1 1254.59,E2 1254.59} C_VEL
LIN {X 0,Y 601.909,Z 611.91,A -85,B 0,C 180,E1 1257.827,E2 1257.827} C_VEL
LIN {X 0,Y 599.463,Z 611.91,A -85,B 0,C 180,E1 1259.056,E2 1259.056} C_VEL
LIN {X 0,Y 593.926,Z 611.91,A -85,B 0,C 180,E1 1260.895,E2 1260.895} C_VEL
LIN {X 0,Y 593.823,Z 611.91,A -85,B 0,C 180,E1 1261.107,E2 1261.107} C_VEL
LIN {X 0,Y 593.832,Z 611.91,A -85,B 0,C 180,E1 1266.09,E2 1266.09} C_VEL
LIN {X 0,Y 593.803,Z 611.91,A -85,B 0,C 180,E1 1270.278,E2 1270.278} C_VEL
LIN {X 0,Y 593.77,Z 611.91,A -85,B 0,C 180,E1 1274.77,E2 1274.77} C_VEL
LIN {X 0,Y 593.887,Z 611.91,A -85,B 0,C 180,E1 1279.391,E2 1279.391} C_VEL
LIN {X 0,Y 593.818,Z 611.91,A -85,B 0,C 180,E1 1284.072,E2 1284.072} C_VEL
LIN {X 0,Y 593.747,Z 611.91,A -85,B 0,C 180,E1 1288.975,E2 1288.975} C_VEL
LIN {X 0,Y 593.858,Z 611.91,A -85,B 0,C 180,E1 1294.113,E2 1294.113} C_VEL
LIN {X 0,Y 593.67,Z 611.91,A -85,B 0,C 180,E1 1300.084,E2 1300.084} C_VEL
LIN {X 0,Y 593.766,Z 611.91,A -85,B 0,C 180,E1 1305.553,E2 1305.553} C_VEL
LIN {X 0,Y 593.731,Z 611.91,A -85,B 0,C 180,E1 1310.393,E2 1310.393} C_VEL
LIN {X 0,Y 593.664,Z 611.91,A -85,B 0,C 180,E1 1315.87,E2 1315.87} C_VEL
LIN {X 0,Y 593.709,Z 611.91,A -85,B 0,C 180,E1 1321.018,E2 1321.018} C_VEL
LIN {X 0,Y 594.005,Z 612.69,A -85,B 0,C 180,E1 1324.011,E2 1324.011} C_VEL
LIN {X 0,Y 596.296,Z 621.582,A -85,B 0,C 180,E1 1324.234,E2 1324.234} C_VEL
LIN {X 0,Y 596.166,Z 669.235,A -85,B 0,C 180,E1 1325.001,E2 1325.001} C_VEL
LIN {X 0,Y 595.967,Z 705.751,A -85,B 0,C 180,E1 1326.185,E2 1326.185} C_VEL
LIN {X 0,Y 595.578,Z 740.146,A -85,B 0,C 180,E1 1327.89,E2 1327.89} C_VEL
LIN {X 0,Y 595.126,Z 772.057,A -85,B 0,C 180,E1 1330.1,E2 1330.1} C_VEL
LIN {X 0,Y 594.747,Z 800.594,A -85,B 0,C 180,E1 1332.768,E2 1332.768} C_VEL
LIN {X 0,Y 594.501,Z 824.392,A -85,B 0,C 180,E1 1335.728,E2 1335.728} C_VEL
LIN {X 0,Y 594.33,Z 843.419,A -85,B 0,C 180,E1 1338.925,E2 1338.925} C_VEL
LIN {X 0,Y 594.26,Z 857.464,A -85,B 0,C 180,E1 1342.313,E2 1342.313} C_VEL
LIN {X 0,Y 594.203,Z 865.973,A -85,B 0,C 180,E1 1345.616,E2 1345.616} C_VEL
LIN {X 0,Y 594.218,Z 869.512,A -85,B 0,C 180,E1 1348.54,E2 1348.54} C_VEL
LIN {X 0,Y 594.305,Z 869.512,A -85,B 0,C 180,E1 1351.46,E2 1351.46} C_VEL
LIN {X 0,Y 594.283,Z 864.448,A -85,B 0,C 180,E1 1355.116,E2 1355.116} C_VEL
LIN {X 0,Y 594.311,Z 854.843,A -85,B 0,C 180,E1 1358.423,E2 1358.423} C_VEL
LIN {X 0,Y 594.432,Z 838.827,A -85,B 0,C 180,E1 1361.944,E2 1361.944} C_VEL
LIN {X 0,Y 594.579,Z 818.198,A -85,B 0,C 180,E1 1365.13,E2 1365.13} C_VEL
LIN {X 0,Y 594.88,Z 793.418,A -85,B 0,C 180,E1 1367.975,E2 1367.975} C_VEL
LIN {X 0,Y 595.291,Z 763.86,A -85,B 0,C 180,E1 1370.535,E2 1370.535} C_VEL
LIN {X 0,Y 595.714,Z 730.011,A -85,B 0,C 180,E1 1372.68,E2 1372.68} C_VEL
LIN {X 0,Y 596.045,Z 694.391,A -85,B 0,C 180,E1 1374.247,E2 1374.247} C_VEL
LIN {X 0,Y 596.32,Z 658.935,A -85,B 0,C 180,E1 1375.218,E2 1375.218} C_VEL
LIN {X 0,Y 595.478,Z 616.641,A -85,B 0,C 180,E1 1375.868,E2 1375.868} C_VEL
LIN {X 0,Y 593.947,Z 611.91,A -85,B 0,C 180,E1 1376.086,E2 1376.086} C_VEL
LIN {X 0,Y 593.859,Z 611.91,A -85,B 0,C 180,E1 1380.657,E2 1380.657} C_VEL
LIN {X 0,Y 593.823,Z 611.91,A -85,B 0,C 180,E1 1385.904,E2 1385.904} C_VEL
LIN {X 0,Y 593.77,Z 611.91,A -85,B 0,C 180,E1 1391.527,E2 1391.527} C_VEL
LIN {X 0,Y 593.657,Z 611.91,A -85,B 0,C 180,E1 1396.486,E2 1396.486} C_VEL
LIN {X 0,Y 593.668,Z 611.91,A -85,B 0,C 180,E1 1402.265,E2 1402.265} C_VEL
LIN {X 0,Y 593.857,Z 611.91,A -85,B 0,C 180,E1 1407.634,E2 1407.634} C_VEL
LIN {X 0,Y 593.735,Z 611.91,A -85,B 0,C 180,E1 1413.191,E2 1413.191} C_VEL
LIN {X 0,Y 593.754,Z 611.91,A -85,B 0,C 180,E1 1417.515,E2 1417.515} C_VEL
LIN {X 0,Y 594.006,Z 611.91,A -85,B 0,C 180,E1 1422.193,E2 1422.193} C_VEL
LIN {X 0,Y 593.918,Z 611.91,A -85,B 0,C 180,E1 1428.236,E2 1428.236} C_VEL
LIN {X 0,Y 593.977,Z 611.91,A -85,B 0,C 180,E1 1432.681,E2 1432.681} C_VEL
LIN {X 0,Y 594.064,Z 611.91,A -85,B 0,C 180,E1 1437.081,E2 1437.081} C_VEL
LIN {X 0,Y 594.2,Z 611.91,A -85,B 0,C 180,E1 1441.463,E2 1441.463} C_VEL
LIN {X 0,Y 594.077,Z 611.91,A -85,B 0,C 180,E1 1446.307,E2 1446.307} C_VEL
LIN {X 0,Y 593.86,Z 611.91,A -85,B 0,C 180,E1 1451.771,E2 1451.771} C_VEL
LIN {X 0,Y 593.89,Z 611.91,A -85,B 0,C 180,E1 1456.288,E2 1456.288} C_VEL
LIN {X 0,Y 593.931,Z 611.91,A -85,B 0,C 180,E1 1460.911,E2 1460.911} C_VEL
LIN {X 0,Y 593.918,Z 611.91,A -85,B 0,C 180,E1 1465.684,E2 1465.684} C_VEL
LIN {X 0,Y 593.771,Z 611.91,A -85,B 0,C 180,E1 1470.664,E2 1470.664} C_VEL
LIN {X 0,Y 593.845,Z 611.91,A -85,B 0,C 180,E1 1475.904,E2 1475.904} C_VEL
LIN {X 0,Y 593.605,Z 611.91,A -85,B 0,C 180,E1 1481.543,E2 1481.543} C_VEL
LIN {X 0,Y 593.787,Z 611.91,A -85,B 0,C 180,E1 1486.492,E2 1486.492} C_VEL
LIN {X 0,Y 593.761,Z 611.91,A -85,B 0,C 180,E1 1492.267,E2 1492.267} C_VEL
LIN {X 0,Y 593.572,Z 611.91,A -85,B 0,C 180,E1 1497.611,E2 1497.611} C_VEL
LIN {X 0,Y 593.707,Z 611.91,A -85,B 0,C 180,E1 1502.675,E2 1502.675} C_VEL
LIN {X 0,Y 593.702,Z 611.91,A -85,B 0,C 180,E1 1507.51,E2 1507.51} C_VEL
LIN {X 0,Y 593.72,Z 611.91,A -85,B 0,C 180,E1 1512.181,E2 1512.181} C_VEL
LIN {X 0,Y 593.762,Z 611.91,A -85,B 0,C 180,E1 1516.733,E2 1516.733} C_VEL
LIN {X 0,Y 593.811,Z 611.91,A -85,B 0,C 180,E1 1521.2,E2 1521.2} C_VEL
LIN {X 0,Y 593.871,Z 611.91,A -85,B 0,C 180,E1 1525.613,E2 1525.613} C_VEL
LIN {X 0,Y 593.956,Z 611.91,A -85,B 0,C 180,E1 1530,E2 1530} C_VEL
LIN {X 0,Y 593.985,Z 611.91,A -85,B 0,C 180,E1 1534.386,E2 1534.386} C_VEL
LIN {X 0,Y 594.042,Z 611.91,A -85,B 0,C 180,E1 1538.796,E2 1538.796} C_VEL
LIN {X 0,Y 593.824,Z 611.91,A -85,B 0,C 180,E1 1544.331,E2 1544.331} C_VEL
LIN {X 0,Y 593.868,Z 611.91,A -85,B 0,C 180,E1 1549.384,E2 1549.384} C_VEL
LIN {X 0,Y 593.769,Z 611.91,A -85,B 0,C 180,E1 1554.078,E2 1554.078} C_VEL
LIN {X 0,Y 593.772,Z 611.91,A -85,B 0,C 180,E1 1558.978,E2 1558.978} C_VEL
LIN {X 0,Y 593.984,Z 611.91,A -85,B 0,C 180,E1 1564.109,E2 1564.109} C_VEL
LIN {X 0,Y 593.721,Z 611.91,A -85,B 0,C 180,E1 1570.089,E2 1570.089} C_VEL
LIN {X 0,Y 593.52,Z 611.91,A -85,B 0,C 180,E1 1575.584,E2 1575.584} C_VEL
LIN {X 0,Y 593.531,Z 611.91,A -85,B 0,C 180,E1 1580.376,E2 1580.376} C_VEL
LIN {X 0,Y 593.634,Z 611.91,A -85,B 0,C 180,E1 1585.866,E2 1585.866} C_VEL
LIN {X 0,Y 593.709,Z 611.91,A -85,B 0,C 180,E1 1591.017,E2 1591.017} C_VEL
LIN {X 0,Y 593.881,Z 611.91,A -85,B 0,C 180,E1 1595.925,E2 1595.925} C_VEL
LIN {X 0,Y 594.03,Z 611.91,A -85,B 0,C 180,E1 1600.648,E2 1600.648} C_VEL
LIN {X 0,Y 593.672,Z 611.91,A -85,B 0,C 180,E1 1605.222,E2 1605.222} C_VEL
LIN {X 0,Y 594.009,Z 611.91,A -85,B 0,C 180,E1 1609.72,E2 1609.72} C_VEL
LIN {X 0,Y 594.233,Z 611.91,A -85,B 0,C 180,E1 1614.148,E2 1614.148} C_VEL
LIN {X 0,Y 593.973,Z 611.91,A -85,B 0,C 180,E1 1619.997,E2 1619.997} C_VEL
LIN {X 0,Y 593.823,Z 611.91,A -85,B 0,C 180,E1 1621.107,E2 1621.107} C_VEL
LIN {X 0,Y 589.923,Z 611.91,A -85,B 0,C 180,E1 1622.761,E2 1622.761} C_VEL
LIN {X 0,Y 586.116,Z 611.91,A -85,B 0,C 180,E1 1624.437,E2 1624.437} C_VEL
LIN {X 0,Y 586.123,Z 611.91,A -85,B 0,C 180,E1 1628.913,E2 1628.913} C_VEL
LIN {X 0,Y 586.155,Z 611.91,A -85,B 0,C 180,E1 1633.439,E2 1633.439} C_VEL
LIN {X 0,Y 585.974,Z 611.91,A -85,B 0,C 180,E1 1639.623,E2 1639.623} C_VEL
LIN {X 0,Y 585.854,Z 611.91,A -85,B 0,C 180,E1 1644.421,E2 1644.421} C_VEL
LIN {X 0,Y 585.774,Z 611.91,A -85,B 0,C 180,E1 1649.408,E2 1649.408} C_VEL
LIN {X 0,Y 585.847,Z 611.91,A -85,B 0,C 180,E1 1654.645,E2 1654.645} C_VEL
LIN {X 0,Y 585.774,Z 611.91,A -85,B 0,C 180,E1 1660.248,E2 1660.248} C_VEL
LIN {X 0,Y 585.897,Z 611.91,A -85,B 0,C 180,E1 1666.343,E2 1666.343} C_VEL
LIN {X 0,Y 585.835,Z 611.91,A -85,B 0,C 180,E1 1671.664,E2 1671.664} C_VEL
LIN {X 0,Y 585.736,Z 611.91,A -85,B 0,C 180,E1 1677.124,E2 1677.124} C_VEL
LIN {X 0,Y 585.797,Z 611.91,A -85,B 0,C 180,E1 1682.783,E2 1682.783} C_VEL
LIN {X 0,Y 585.99,Z 611.91,A -85,B 0,C 180,E1 1683.614,E2 1683.614} C_VEL
LIN {X 0,Y 589.176,Z 621.679,A -85,B 0,C 180,E1 1683.901,E2 1683.901} C_VEL
LIN {X 0,Y 588.994,Z 671.019,A -85,B 0,C 180,E1 1684.721,E2 1684.721} C_VEL
LIN {X 0,Y 588.674,Z 707.137,A -85,B 0,C 180,E1 1685.929,E2 1685.929} C_VEL
LIN {X 0,Y 588.11,Z 742.077,A -85,B 0,C 180,E1 1687.708,E2 1687.708} C_VEL
LIN {X 0,Y 587.533,Z 774.003,A -85,B 0,C 180,E1 1689.995,E2 1689.995} C_VEL
LIN {X 0,Y 587.01,Z 802.462,A -85,B 0,C 180,E1 1692.739,E2 1692.739} C_VEL
LIN {X 0,Y 586.645,Z 827.203,A -85,B 0,C 180,E1 1695.95,E2 1695.95} C_VEL
LIN {X 0,Y 586.432,Z 845.363,A -85,B 0,C 180,E1 1699.189,E2 1699.189} C_VEL
LIN {X 0,Y 586.37,Z 858.615,A -85,B 0,C 180,E1 1702.582,E2 1702.582} C_VEL
LIN {X 0,Y 586.328,Z 867.17,A -85,B 0,C 180,E1 1706.299,E2 1706.299} C_VEL
LIN {X 0,Y 586.296,Z 870,A -85,B 0,C 180,E1 1710,E2 1710} C_VEL
LIN {X 0,Y 586.389,Z 867.17,A -85,B 0,C 180,E1 1713.701,E2 1713.701} C_VEL
LIN {X 0,Y 586.41,Z 858.615,A -85,B 0,C 180,E1 1717.417,E2 1717.417} C_VEL
LIN {X 0,Y 586.53,Z 845.261,A -85,B 0,C 180,E1 1720.831,E2 1720.831} C_VEL
LIN {X 0,Y 586.735,Z 826.078,A -85,B 0,C 180,E1 1724.221,E2 1724.221} C_VEL
LIN {X 0,Y 587.093,Z 800.946,A -85,B 0,C 180,E1 1727.425,E2 1727.425} C_VEL
LIN {X 0,Y 587.566,Z 772.296,A -85,B 0,C 180,E1 1730.146,E2 1730.146} C_VEL
LIN {X 0,Y 588.129,Z 739.934,A -85,B 0,C 180,E1 1732.418,E2 1732.418} C_VEL
LIN {X 0,Y 588.586,Z 705.103,A -85,B 0,C 180,E1 1734.16,E2 1734.16} C_VEL
LIN {X 0,Y 588.987,Z 668.059,A -85,B 0,C 180,E1 1735.355,E2 1735.355} C_VEL
LIN {X 0,Y 588.543,Z 619.451,A -85,B 0,C 180,E1 1736.159,E2 1736.159} C_VEL
LIN {X 0,Y 585.967,Z 611.91,A -85,B 0,C 180,E1 1736.469,E2 1736.469} C_VEL
LIN {X 0,Y 585.812,Z 611.91,A -85,B 0,C 180,E1 1741.481,E2 1741.481} C_VEL
LIN {X 0,Y 585.845,Z 611.91,A -85,B 0,C 180,E1 1746.766,E2 1746.766} C_VEL
LIN {X 0,Y 585.878,Z 611.91,A -85,B 0,C 180,E1 1752.214,E2 1752.214} C_VEL
LIN {X 0,Y 585.691,Z 611.91,A -85,B 0,C 180,E1 1757.775,E2 1757.775} C_VEL
LIN {X 0,Y 585.682,Z 611.91,A -85,B 0,C 180,E1 1763.263,E2 1763.263} C_VEL
LIN {X 0,Y 585.898,Z 611.91,A -85,B 0,C 180,E1 1768.515,E2 1768.515} C_VEL
LIN {X 0,Y 585.804,Z 611.91,A -85,B 0,C 180,E1 1773.94,E2 1773.94} C_VEL
LIN {X 0,Y 585.772,Z 611.91,A -85,B 0,C 180,E1 1778.789,E2 1778.789} C_VEL
LIN {X 0,Y 585.93,Z 611.91,A -85,B 0,C 180,E1 1783.49,E2 1783.49} C_VEL
LIN {X 0,Y 586.038,Z 611.91,A -85,B 0,C 180,E1 1788.075,E2 1788.075} C_VEL
LIN {X 0,Y 586.071,Z 611.91,A -85,B 0,C 180,E1 1792.581,E2 1792.581} C_VEL
LIN {X 0,Y 586.171,Z 611.91,A -85,B 0,C 180,E1 1797.042,E2 1797.042} C_VEL
LIN {X 0,Y 586.299,Z 611.91,A -85,B 0,C 180,E1 1801.482,E2 1801.482} C_VEL
LIN {X 0,Y 586.311,Z 611.91,A -85,B 0,C 180,E1 1805.931,E2 1805.931} C_VEL
LIN {X 0,Y 585.928,Z 611.91,A -85,B 0,C 180,E1 1811.933,E2 1811.933} C_VEL
LIN {X 0,Y 585.861,Z 611.91,A -85,B 0,C 180,E1 1817.02,E2 1817.02} C_VEL
LIN {X 0,Y 585.914,Z 611.91,A -85,B 0,C 180,E1 1821.523,E2 1821.523} C_VEL
LIN {X 0,Y 585.957,Z 611.91,A -85,B 0,C 180,E1 1826.059,E2 1826.059} C_VEL
LIN {X 0,Y 585.746,Z 611.91,A -85,B 0,C 180,E1 1831.461,E2 1831.461} C_VEL
LIN {X 0,Y 585.921,Z 611.91,A -85,B 0,C 180,E1 1836.769,E2 1836.769} C_VEL
LIN {X 0,Y 585.708,Z 611.91,A -85,B 0,C 180,E1 1842.231,E2 1842.231} C_VEL
LIN {X 0,Y 585.872,Z 611.91,A -85,B 0,C 180,E1 1847.785,E2 1847.785} C_VEL
LIN {X 0,Y 585.815,Z 611.91,A -85,B 0,C 180,E1 1853.527,E2 1853.527} C_VEL
LIN {X 0,Y 585.757,Z 611.91,A -85,B 0,C 180,E1 1858.872,E2 1858.872} C_VEL
LIN {X 0,Y 586.003,Z 611.91,A -85,B 0,C 180,E1 1864.73,E2 1864.73} C_VEL
LIN {X 0,Y 585.974,Z 611.91,A -85,B 0,C 180,E1 1870.373,E2 1870.373} C_VEL
LIN {X 0,Y 586.053,Z 611.91,A -85,B 0,C 180,E1 1875.028,E2 1875.028} C_VEL
LIN {X 0,Y 586.096,Z 611.91,A -85,B 0,C 180,E1 1879.582,E2 1879.582} C_VEL
LIN {X 0,Y 586.281,Z 611.91,A -85,B 0,C 180,E1 1884.071,E2 1884.071} C_VEL
LIN {X 0,Y 586.067,Z 611.91,A -85,B 0,C 180,E1 1890,E2 1890} C_VEL
LIN {X 0,Y 586.08,Z 611.91,A -85,B 0,C 180,E1 1894.445,E2 1894.445} C_VEL
LIN {X 0,Y 586.105,Z 611.91,A -85,B 0,C 180,E1 1898.916,E2 1898.916} C_VEL
LIN {X 0,Y 586.136,Z 611.91,A -85,B 0,C 180,E1 1903.443,E2 1903.443} C_VEL
LIN {X 0,Y 585.955,Z 611.91,A -85,B 0,C 180,E1 1909.628,E2 1909.628} C_VEL
LIN {X 0,Y 585.786,Z 611.91,A -85,B 0,C 180,E1 1915.225,E2 1915.225} C_VEL
LIN {X 0,Y 585.809,Z 611.91,A -85,B 0,C 180,E1 1919.411,E2 1919.411} C_VEL
LIN {X 0,Y 586.023,Z 611.91,A -85,B 0,C 180,E1 1924.638,E2 1924.638} C_VEL
LIN {X 0,Y 585.833,Z 611.91,A -85,B 0,C 180,E1 1930.249,E2 1930.249} C_VEL
LIN {X 0,Y 585.699,Z 611.91,A -85,B 0,C 180,E1 1936.37,E2 1936.37} C_VEL
LIN {X 0,Y 585.661,Z 611.91,A -85,B 0,C 180,E1 1941.649,E2 1941.649} C_VEL
LIN {X 0,Y 585.692,Z 611.91,A -85,B 0,C 180,E1 1947.119,E2 1947.119} C_VEL
LIN {X 0,Y 585.751,Z 611.91,A -85,B 0,C 180,E1 1952.271,E2 1952.271} C_VEL
LIN {X 0,Y 585.846,Z 611.91,A -85,B 0,C 180,E1 1957.189,E2 1957.189} C_VEL
LIN {X 0,Y 586.087,Z 611.91,A -85,B 0,C 180,E1 1961.939,E2 1961.939} C_VEL
LIN {X 0,Y 585.766,Z 611.91,A -85,B 0,C 180,E1 1968.064,E2 1968.064} C_VEL
LIN {X 0,Y 586.312,Z 611.91,A -85,B 0,C 180,E1 1974.069,E2 1974.069} C_VEL
LIN {X 0,Y 586.083,Z 611.91,A -85,B 0,C 180,E1 1979.997,E2 1979.997} C_VEL
LIN {X 0,Y 586.116,Z 611.91,A -85,B 0,C 180,E1 1984.437,E2 1984.437} C_VEL
LIN {X 0,Y 583.648,Z 611.91,A -85,B 0,C 180,E1 1985.694,E2 1985.694} C_VEL
LIN {X 0,Y 578.246,Z 611.91,A -85,B 0,C 180,E1 1987.575,E2 1987.575} C_VEL
LIN {X 0,Y 578.14,Z 611.91,A -85,B 0,C 180,E1 1987.793,E2 1987.793} C_VEL
LIN {X 0,Y 578.193,Z 611.91,A -85,B 0,C 180,E1 1993.628,E2 1993.628} C_VEL
LIN {X 0,Y 578.081,Z 611.91,A -85,B 0,C 180,E1 1999.459,E2 1999.459} C_VEL
LIN {X 0,Y 577.945,Z 611.91,A -85,B 0,C 180,E1 2004.777,E2 2004.777} C_VEL
LIN {X 0,Y 577.805,Z 611.91,A -85,B 0,C 180,E1 2010.15,E2 2010.15} C_VEL
LIN {X 0,Y 577.828,Z 611.91,A -85,B 0,C 180,E1 2015.197,E2 2015.197} C_VEL
LIN {X 0,Y 577.815,Z 611.91,A -85,B 0,C 180,E1 2020.92,E2 2020.92} C_VEL
LIN {X 0,Y 577.949,Z 611.91,A -85,B 0,C 180,E1 2027.069,E2 2027.069} C_VEL
LIN {X 0,Y 577.953,Z 611.91,A -85,B 0,C 180,E1 2032.949,E2 2032.949} C_VEL
LIN {X 0,Y 577.906,Z 611.91,A -85,B 0,C 180,E1 2038.4,E2 2038.4} C_VEL
LIN {X 0,Y 578,Z 611.91,A -85,B 0,C 180,E1 2043.215,E2 2043.215} C_VEL
LIN {X 0,Y 582.112,Z 624.656,A -85,B 0,C 180,E1 2043.6,E2 2043.6} C_VEL
LIN {X 0,Y 581.837,Z 671.039,A -85,B 0,C 180,E1 2044.388,E2 2044.388} C_VEL
LIN {X 0,Y 581.38,Z 708.113,A -85,B 0,C 180,E1 2045.65,E2 2045.65} C_VEL
LIN {X 0,Y 580.703,Z 742.075,A -85,B 0,C 180,E1 2047.408,E2 2047.408} C_VEL
LIN {X 0,Y 579.926,Z 774.485,A -85,B 0,C 180,E1 2049.762,E2 2049.762} C_VEL
LIN {X 0,Y 579.31,Z 802.467,A -85,B 0,C 180,E1 2052.503,E2 2052.503} C_VEL
LIN {X 0,Y 578.861,Z 826.818,A -85,B 0,C 180,E1 2055.695,E2 2055.695} C_VEL
LIN {X 0,Y 578.597,Z 845.362,A -85,B 0,C 180,E1 2059.041,E2 2059.041} C_VEL
LIN {X 0,Y 578.501,Z 858.619,A -85,B 0,C 180,E1 2062.481,E2 2062.481} C_VEL
LIN {X 0,Y 578.447,Z 867.172,A -85,B 0,C 180,E1 2066.248,E2 2066.248} C_VEL
LIN {X 0,Y 578.396,Z 870,A -85,B 0,C 180,E1 2070,E2 2070} C_VEL
LIN {X 0,Y 578.512,Z 867.172,A -85,B 0,C 180,E1 2073.751,E2 2073.751} C_VEL
LIN {X 0,Y 578.539,Z 858.619,A -85,B 0,C 180,E1 2077.519,E2 2077.519} C_VEL
LIN {X 0,Y 578.687,Z 845.26,A -85,B 0,C 180,E1 2080.98,E2 2080.98} C_VEL
LIN {X 0,Y 578.972,Z 825.413,A -85,B 0,C 180,E1 2084.512,E2 2084.512} C_VEL
LIN {X 0,Y 579.408,Z 800.951,A -85,B 0,C 180,E1 2087.664,E2 2087.664} C_VEL
LIN {X 0,Y 580.045,Z 771.862,A -85,B 0,C 180,E1 2090.454,E2 2090.454} C_VEL
LIN {X 0,Y 580.699,Z 740.396,A -85,B 0,C 180,E1 2092.693,E2 2092.693} C_VEL
LIN {X 0,Y 581.322,Z 705.076,A -85,B 0,C 180,E1 2094.483,E2 2094.483} C_VEL
LIN {X 0,Y 581.835,Z 668.024,A -85,B 0,C 180,E1 2095.689,E2 2095.689} C_VEL
LIN {X 0,Y 581.429,Z 621.666,A -85,B 0,C 180,E1 2096.474,E2 2096.474} C_VEL
LIN {X 0,Y 577.998,Z 611.91,A -85,B 0,C 180,E1 2096.864,E2 2096.864} C_VEL
LIN {X 0,Y 577.905,Z 611.91,A -85,B 0,C 180,E1 2101.6,E2 2101.6} C_VEL
LIN {X 0,Y 577.926,Z 611.91,A -85,B 0,C 180,E1 2107.053,E2 2107.053} C_VEL
LIN {X 0,Y 577.934,Z 611.91,A -85,B 0,C 180,E1 2112.933,E2 2112.933} C_VEL
LIN {X 0,Y 577.799,Z 611.91,A -85,B 0,C 180,E1 2119.079,E2 2119.079} C_VEL
LIN {X 0,Y 577.827,Z 611.91,A -85,B 0,C 180,E1 2124.803,E2 2124.803} C_VEL
LIN {X 0,Y 577.956,Z 611.91,A -85,B 0,C 180,E1 2130.154,E2 2130.154} C_VEL
LIN {X 0,Y 577.921,Z 611.91,A -85,B 0,C 180,E1 2135.222,E2 2135.222} C_VEL
LIN {X 0,Y 577.983,Z 611.91,A -85,B 0,C 180,E1 2140.568,E2 2140.568} C_VEL
LIN {X 0,Y 578.181,Z 611.91,A -85,B 0,C 180,E1 2146.372,E2 2146.372} C_VEL
LIN {X 0,Y 578.172,Z 611.91,A -85,B 0,C 180,E1 2152.479,E2 2152.479} C_VEL
LIN {X 0,Y 578.263,Z 611.91,A -85,B 0,C 180,E1 2157.001,E2 2157.001} C_VEL
LIN {X 0,Y 578.389,Z 611.91,A -85,B 0,C 180,E1 2161.503,E2 2161.503} C_VEL
LIN {X 0,Y 578.395,Z 611.91,A -85,B 0,C 180,E1 2166.013,E2 2166.013} C_VEL
LIN {X 0,Y 578.005,Z 611.91,A -85,B 0,C 180,E1 2172.099,E2 2172.099} C_VEL
LIN {X 0,Y 578.017,Z 611.91,A -85,B 0,C 180,E1 2176.748,E2 2176.748} C_VEL
LIN {X 0,Y 578.025,Z 611.91,A -85,B 0,C 180,E1 2181.515,E2 2181.515} C_VEL
LIN {X 0,Y 577.897,Z 611.91,A -85,B 0,C 180,E1 2187.029,E2 2187.029} C_VEL
LIN {X 0,Y 577.812,Z 611.91,A -85,B 0,C 180,E1 2193.018,E2 2193.018} C_VEL
LIN {X 0,Y 577.98,Z 611.91,A -85,B 0,C 180,E1 2198.956,E2 2198.956} C_VEL
LIN {X 0,Y 577.917,Z 611.91,A -85,B 0,C 180,E1 2205.022,E2 2205.022} C_VEL
LIN {X 0,Y 577.851,Z 611.91,A -85,B 0,C 180,E1 2211.036,E2 2211.036} C_VEL
LIN {X 0,Y 577.793,Z 611.91,A -85,B 0,C 180,E1 2216.987,E2 2216.987} C_VEL
LIN {X 0,Y 577.915,Z 611.91,A -85,B 0,C 180,E1 2222.969,E2 2222.969} C_VEL
LIN {X 0,Y 578.017,Z 611.91,A -85,B 0,C 180,E1 2228.487,E2 2228.487} C_VEL
LIN {X 0,Y 578.127,Z 611.91,A -85,B 0,C 180,E1 2234.818,E2 2234.818} C_VEL
LIN {X 0,Y 578.029,Z 611.91,A -85,B 0,C 180,E1 2240.958,E2 2240.958} C_VEL
LIN {X 0,Y 578.096,Z 611.91,A -85,B 0,C 180,E1 2245.494,E2 2245.494} C_VEL
LIN {X 0,Y 578.166,Z 611.91,A -85,B 0,C 180,E1 2250,E2 2250} C_VEL
LIN {X 0,Y 578.166,Z 611.91,A -85,B 0,C 180,E1 2254.506,E2 2254.506} C_VEL
LIN {X 0,Y 578.174,Z 611.91,A -85,B 0,C 180,E1 2259.04,E2 2259.04} C_VEL
LIN {X 0,Y 578.034,Z 611.91,A -85,B 0,C 180,E1 2264.268,E2 2264.268} C_VEL
LIN {X 0,Y 578.027,Z 611.91,A -85,B 0,C 180,E1 2269.908,E2 2269.908} C_VEL
LIN {X 0,Y 577.919,Z 611.91,A -85,B 0,C 180,E1 2274.782,E2 2274.782} C_VEL
LIN {X 0,Y 577.857,Z 611.91,A -85,B 0,C 180,E1 2280.157,E2 2280.157} C_VEL
LIN {X 0,Y 578.014,Z 611.91,A -85,B 0,C 180,E1 2285.189,E2 2285.189} C_VEL
LIN {X 0,Y 577.895,Z 611.91,A -85,B 0,C 180,E1 2290.919,E2 2290.919} C_VEL
LIN {X 0,Y 577.82,Z 611.91,A -85,B 0,C 180,E1 2297.196,E2 2297.196} C_VEL
LIN {X 0,Y 577.834,Z 611.91,A -85,B 0,C 180,E1 2302.938,E2 2302.938} C_VEL
LIN {X 0,Y 577.846,Z 611.91,A -85,B 0,C 180,E1 2308.395,E2 2308.395} C_VEL
LIN {X 0,Y 577.971,Z 611.91,A -85,B 0,C 180,E1 2313.554,E2 2313.554} C_VEL
LIN {X 0,Y 578.047,Z 611.91,A -85,B 0,C 180,E1 2318.486,E2 2318.486} C_VEL
LIN {X 0,Y 578.196,Z 611.91,A -85,B 0,C 180,E1 2323.257,E2 2323.257} C_VEL
LIN {X 0,Y 578.134,Z 611.91,A -85,B 0,C 180,E1 2329.434,E2 2329.434} C_VEL
LIN {X 0,Y 578.397,Z 611.91,A -85,B 0,C 180,E1 2334.107,E2 2334.107} C_VEL
LIN {X 0,Y 578.182,Z 611.91,A -85,B 0,C 180,E1 2339.997,E2 2339.997} C_VEL
LIN {X 0,Y 578.201,Z 611.91,A -85,B 0,C 180,E1 2344.503,E2 2344.503} C_VEL
LIN {X 0,Y 578.14,Z 611.91,A -85,B 0,C 180,E1 2347.793,E2 2347.793} C_VEL
LIN {X 0,Y 576.837,Z 611.91,A -85,B 0,C 180,E1 2348.648,E2 2348.648} C_VEL
LIN {X 0,Y 570.206,Z 611.91,A -85,B 0,C 180,E1 2350.974,E2 2350.974} C_VEL
LIN {X 0,Y 570.116,Z 611.91,A -85,B 0,C 180,E1 2351.195,E2 2351.195} C_VEL
LIN {X 0,Y 570.031,Z 611.91,A -85,B 0,C 180,E1 2355.4,E2 2355.4} C_VEL
LIN {X 0,Y 570.104,Z 611.91,A -85,B 0,C 180,E1 2360.193,E2 2360.193} C_VEL
LIN {X 0,Y 569.97,Z 611.91,A -85,B 0,C 180,E1 2365.423,E2 2365.423} C_VEL
LIN {X 0,Y 569.921,Z 611.91,A -85,B 0,C 180,E1 2370.31,E2 2370.31} C_VEL
LIN {X 0,Y 569.889,Z 611.91,A -85,B 0,C 180,E1 2375.762,E2 2375.762} C_VEL
LIN {X 0,Y 569.841,Z 611.91,A -85,B 0,C 180,E1 2381.619,E2 2381.619} C_VEL
LIN {X 0,Y 569.955,Z 611.91,A -85,B 0,C 180,E1 2386.316,E2 2386.316} C_VEL
LIN {X 0,Y 570.035,Z 611.91,A -85,B 0,C 180,E1 2392.346,E2 2392.346} C_VEL
LIN {X 0,Y 569.99,Z 611.91,A -85,B 0,C 180,E1 2398.204,E2 2398.204} C_VEL
LIN {X 0,Y 570.02,Z 611.91,A -85,B 0,C 180,E1 2402.789,E2 2402.789} C_VEL
LIN {X 0,Y 575.029,Z 625.572,A -85,B 0,C 180,E1 2403.262,E2 2403.262} C_VEL
LIN {X 0,Y 574.678,Z 672.239,A -85,B 0,C 180,E1 2404.077,E2 2404.077} C_VEL
LIN {X 0,Y 574.065,Z 709.645,A -85,B 0,C 180,E1 2405.387,E2 2405.387} C_VEL
LIN {X 0,Y 573.222,Z 744.141,A -85,B 0,C 180,E1 2407.232,E2 2407.232} C_VEL
LIN {X 0,Y 572.339,Z 776.021,A -85,B 0,C 180,E1 2409.618,E2 2409.618} C_VEL
LIN {X 0,Y 571.55,Z 804.296,A -85,B 0,C 180,E1 2412.471,E2 2412.471} C_VEL
LIN {X 0,Y 571.027,Z 828.417,A -85,B 0,C 180,E1 2415.753,E2 2415.753} C_VEL
LIN {X 0,Y 570.725,Z 845.655,A -85,B 0,C 180,E1 2418.953,E2 2418.953} C_VEL
LIN {X 0,Y 570.611,Z 858.622,A -85,B 0,C 180,E1 2422.376,E2 2422.376} C_VEL
LIN {X 0,Y 570.544,Z 867.173,A -85,B 0,C 180,E1 2426.196,E2 2426.196} C_VEL
LIN {X 0,Y 570.497,Z 870,A -85,B 0,C 180,E1 2430,E2 2430} C_VEL
LIN {X 0,Y 570.612,Z 867.173,A -85,B 0,C 180,E1 2433.804,E2 2433.804} C_VEL
LIN {X 0,Y 570.65,Z 858.622,A -85,B 0,C 180,E1 2437.623,E2 2437.623} C_VEL
LIN {X 0,Y 570.851,Z 844.805,A -85,B 0,C 180,E1 2441.232,E2 2441.232} C_VEL
LIN {X 0,Y 571.192,Z 825.408,A -85,B 0,C 180,E1 2444.714,E2 2444.714} C_VEL
LIN {X 0,Y 571.712,Z 800.978,A -85,B 0,C 180,E1 2447.907,E2 2447.907} C_VEL
LIN {X 0,Y 572.478,Z 772.102,A -85,B 0,C 180,E1 2450.716,E2 2450.716} C_VEL
LIN {X 0,Y 573.311,Z 740.181,A -85,B 0,C 180,E1 2453.015,E2 2453.015} C_VEL
LIN {X 0,Y 574.124,Z 703.789,A -85,B 0,C 180,E1 2454.866,E2 2454.866} C_VEL
LIN {X 0,Y 574.718,Z 666.563,A -85,B 0,C 180,E1 2456.064,E2 2456.064} C_VEL
LIN {X 0,Y 574.429,Z 623.748,A -85,B 0,C 180,E1 2456.793,E2 2456.793} C_VEL
LIN {X 0,Y 570.034,Z 611.91,A -85,B 0,C 180,E1 2457.215,E2 2457.215} C_VEL
LIN {X 0,Y 569.956,Z 611.91,A -85,B 0,C 180,E1 2462.093,E2 2462.093} C_VEL
LIN {X 0,Y 570.01,Z 611.91,A -85,B 0,C 180,E1 2467.656,E2 2467.656} C_VEL
LIN {X 0,Y 569.942,Z 611.91,A -85,B 0,C 180,E1 2473.685,E2 2473.685} C_VEL
LIN {X 0,Y 569.827,Z 611.91,A -85,B 0,C 180,E1 2478.38,E2 2478.38} C_VEL
LIN {X 0,Y 569.887,Z 611.91,A -85,B 0,C 180,E1 2484.238,E2 2484.238} C_VEL
LIN {X 0,Y 570.063,Z 611.91,A -85,B 0,C 180,E1 2489.698,E2 2489.698} C_VEL
LIN {X 0,Y 569.967,Z 611.91,A -85,B 0,C 180,E1 2494.852,E2 2494.852} C_VEL
LIN {X 0,Y 570.006,Z 611.91,A -85,B 0,C 180,E1 2499.803,E2 2499.803} C_VEL
LIN {X 0,Y 570.034,Z 611.91,A -85,B 0,C 180,E1 2504.6,E2 2504.6} C_VEL
LIN {X 0,Y 570.132,Z 611.91,A -85,B 0,C 180,E1 2509.29,E2 2509.29} C_VEL
LIN {X 0,Y 570.175,Z 611.91,A -85,B 0,C 180,E1 2513.906,E2 2513.906} C_VEL
LIN {X 0,Y 570.185,Z 611.91,A -85,B 0,C 180,E1 2518.481,E2 2518.481} C_VEL
LIN {X 0,Y 570.199,Z 611.91,A -85,B 0,C 180,E1 2523.047,E2 2523.047} C_VEL
LIN {X 0,Y 570.136,Z 611.91,A -85,B 0,C 180,E1 2527.633,E2 2527.633} C_VEL
LIN {X 0,Y 570.102,Z 611.91,A -85,B 0,C 180,E1 2532.269,E2 2532.269} C_VEL
LIN {X 0,Y 570.08,Z 611.91,A -85,B 0,C 180,E1 2537.038,E2 2537.038} C_VEL
LIN {X 0,Y 570.073,Z 611.91,A -85,B 0,C 180,E1 2541.83,E2 2541.83} C_VEL
LIN {X 0,Y 570.011,Z 611.91,A -85,B 0,C 180,E1 2546.845,E2 2546.845} C_VEL
LIN {X 0,Y 569.903,Z 611.91,A -85,B 0,C 180,E1 2552.098,E2 2552.098} C_VEL
LIN {X 0,Y 570.105,Z 611.91,A -85,B 0,C 180,E1 2557.651,E2 2557.651} C_VEL
LIN {X 0,Y 569.895,Z 611.91,A -85,B 0,C 180,E1 2564.167,E2 2564.167} C_VEL
LIN {X 0,Y 569.944,Z 611.91,A -85,B 0,C 180,E1 2568.385,E2 2568.385} C_VEL
LIN {X 0,Y 569.94,Z 611.91,A -85,B 0,C 180,E1 2574.237,E2 2574.237} C_VEL
LIN {X 0,Y 569.959,Z 611.91,A -85,B 0,C 180,E1 2579.687,E2 2579.687} C_VEL
LIN {X 0,Y 570.121,Z 611.91,A -85,B 0,C 180,E1 2584.855,E2 2584.855} C_VEL
LIN {X 0,Y 570.11,Z 611.91,A -85,B 0,C 180,E1 2589.803,E2 2589.803} C_VEL
LIN {X 0,Y 570.186,Z 611.91,A -85,B 0,C 180,E1 2594.601,E2 2594.601} C_VEL
LIN {X 0,Y 570.247,Z 611.91,A -85,B 0,C 180,E1 2599.289,E2 2599.289} C_VEL
LIN {X 0,Y 570.43,Z 611.91,A -85,B 0,C 180,E1 2603.905,E2 2603.905} C_VEL
LIN {X 0,Y 570.28,Z 611.91,A -85,B 0,C 180,E1 2610,E2 2610} C_VEL
LIN {X 0,Y 570.267,Z 611.91,A -85,B 0,C 180,E1 2614.568,E2 2614.568} C_VEL
LIN {X 0,Y 570.242,Z 611.91,A -85,B 0,C 180,E1 2619.167,E2 2619.167} C_VEL
LIN {X 0,Y 570.237,Z 611.91,A -85,B 0,C 180,E1 2623.825,E2 2623.825} C_VEL
LIN {X 0,Y 570.196,Z 611.91,A -85,B 0,C 180,E1 2628.581,E2 2628.581} C_VEL
LIN {X 0,Y 570.094,Z 611.91,A -85,B 0,C 180,E1 2633.476,E2 2633.476} C_VEL
LIN {X 0,Y 569.992,Z 611.91,A -85,B 0,C 180,E1 2638.767,E2 2638.767} C_VEL
LIN {X 0,Y 570.114,Z 611.91,A -85,B 0,C 180,E1 2644.585,E2 2644.585} C_VEL
LIN {X 0,Y 569.993,Z 611.91,A -85,B 0,C 180,E1 2649.616,E2 2649.616} C_VEL
LIN {X 0,Y 569.755,Z 611.91,A -85,B 0,C 180,E1 2655.848,E2 2655.848} C_VEL
LIN {X 0,Y 569.785,Z 611.91,A -85,B 0,C 180,E1 2660.408,E2 2660.408} C_VEL
LIN {X 0,Y 569.845,Z 611.91,A -85,B 0,C 180,E1 2665.453,E2 2665.453} C_VEL
LIN {X 0,Y 569.933,Z 611.91,A -85,B 0,C 180,E1 2671.242,E2 2671.242} C_VEL
LIN {X 0,Y 570.077,Z 611.91,A -85,B 0,C 180,E1 2676.521,E2 2676.521} C_VEL
LIN {X 0,Y 570.254,Z 611.91,A -85,B 0,C 180,E1 2681.419,E2 2681.419} C_VEL
LIN {X 0,Y 569.815,Z 611.91,A -85,B 0,C 180,E1 2686.162,E2 2686.162} C_VEL
LIN {X 0,Y 570.096,Z 611.91,A -85,B 0,C 180,E1 2691.388,E2 2691.388} C_VEL
LIN {X 0,Y 570.249,Z 611.91,A -85,B 0,C 180,E1 2695.429,E2 2695.429} C_VEL
LIN {X 0,Y 570.294,Z 611.91,A -85,B 0,C 180,E1 2699.997,E2 2699.997} C_VEL
LIN {X 0,Y 570.3,Z 611.91,A -85,B 0,C 180,E1 2704.565,E2 2704.565} C_VEL
LIN {X 0,Y 570.258,Z 611.91,A -85,B 0,C 180,E1 2709.163,E2 2709.163} C_VEL
LIN {X 0,Y 570.116,Z 611.91,A -85,B 0,C 180,E1 2711.195,E2 2711.195} C_VEL
LIN {X 0,Y 568.894,Z 611.91,A -85,B 0,C 180,E1 2712.062,E2 2712.062} C_VEL
LIN {X 0,Y 562.187,Z 611.91,A -85,B 0,C 180,E1 2714.648,E2 2714.648} C_VEL
LIN {X 0,Y 562.2,Z 611.91,A -85,B 0,C 180,E1 2720.49,E2 2720.49} C_VEL
LIN {X 0,Y 562.074,Z 611.91,A -85,B 0,C 180,E1 2725.526,E2 2725.526} C_VEL
LIN {X 0,Y 562.008,Z 611.91,A -85,B 0,C 180,E1 2730.783,E2 2730.783} C_VEL
LIN {X 0,Y 561.978,Z 611.91,A -85,B 0,C 180,E1 2736.345,E2 2736.345} C_VEL
LIN {X 0,Y 561.914,Z 611.91,A -85,B 0,C 180,E1 2742.341,E2 2742.341} C_VEL
LIN {X 0,Y 562.036,Z 611.91,A -85,B 0,C 180,E1 2747.665,E2 2747.665} C_VEL
LIN {X 0,Y 562.089,Z 611.91,A -85,B 0,C 180,E1 2753.901,E2 2753.901} C_VEL
LIN {X 0,Y 562.105,Z 611.91,A -85,B 0,C 180,E1 2759.525,E2 2759.525} C_VEL
LIN {X 0,Y 562.083,Z 611.91,A -85,B 0,C 180,E1 2762.37,E2 2762.37} C_VEL
LIN {X 0,Y 567.988,Z 628.975,A -85,B 0,C 180,E1 2762.951,E2 2762.951} C_VEL
LIN {X 0,Y 567.559,Z 672.259,A -85,B 0,C 180,E1 2763.727,E2 2763.727} C_VEL
LIN {X 0,Y 566.84,Z 709.582,A -85,B 0,C 180,E1 2765.05,E2 2765.05} C_VEL
LIN {X 0,Y 565.886,Z 742.721,A -85,B 0,C 180,E1 2766.824,E2 2766.824} C_VEL
LIN {X 0,Y 564.779,Z 775.628,A -85,B 0,C 180,E1 2769.297,E2 2769.297} C_VEL
LIN {X 0,Y 563.867,Z 804.288,A -85,B 0,C 180,E1 2772.224,E2 2772.224} C_VEL
LIN {X 0,Y 563.275,Z 827.301,A -85,B 0,C 180,E1 2775.369,E2 2775.369} C_VEL
LIN {X 0,Y 562.88,Z 845.654,A -85,B 0,C 180,E1 2778.797,E2 2778.797} C_VEL
LIN {X 0,Y 562.734,Z 858.626,A -85,B 0,C 180,E1 2782.269,E2 2782.269} C_VEL
LIN {X 0,Y 562.649,Z 865.977,A -85,B 0,C 180,E1 2785.37,E2 2785.37} C_VEL
LIN {X 0,Y 562.623,Z 869.523,A -85,B 0,C 180,E1 2788.458,E2 2788.458} C_VEL
LIN {X 0,Y 562.693,Z 869.523,A -85,B 0,C 180,E1 2791.542,E2 2791.542} C_VEL
LIN {X 0,Y 562.684,Z 864.367,A -85,B 0,C 180,E1 2795.44,E2 2795.44} C_VEL
LIN {X 0,Y 562.777,Z 854.857,A -85,B 0,C 180,E1 2798.899,E2 2798.899} C_VEL
LIN {X 0,Y 563.008,Z 838.805,A -85,B 0,C 180,E1 2802.621,E2 2802.621} C_VEL
LIN {X 0,Y 563.487,Z 818.199,A -85,B 0,C 180,E1 2805.987,E2 2805.987} C_VEL
LIN {X 0,Y 564.262,Z 791.971,A -85,B 0,C 180,E1 2809.14,E2 2809.14} C_VEL
LIN {X 0,Y 565.254,Z 762.053,A -85,B 0,C 180,E1 2811.817,E2 2811.817} C_VEL
LIN {X 0,Y 566.328,Z 729.033,A -85,B 0,C 180,E1 2813.984,E2 2813.984} C_VEL
LIN {X 0,Y 567.216,Z 694.525,A -85,B 0,C 180,E1 2815.56,E2 2815.56} C_VEL
LIN {X 0,Y 567.859,Z 659.579,A -85,B 0,C 180,E1 2816.566,E2 2816.566} C_VEL
LIN {X 0,Y 567.609,Z 626.603,A -85,B 0,C 180,E1 2817.102,E2 2817.102} C_VEL
LIN {X 0,Y 562.091,Z 611.91,A -85,B 0,C 180,E1 2817.63,E2 2817.63} C_VEL
LIN {X 0,Y 561.945,Z 611.91,A -85,B 0,C 180,E1 2823.368,E2 2823.368} C_VEL
LIN {X 0,Y 562.026,Z 611.91,A -85,B 0,C 180,E1 2828.633,E2 2828.633} C_VEL
LIN {X 0,Y 562.02,Z 611.91,A -85,B 0,C 180,E1 2834.461,E2 2834.461} C_VEL
LIN {X 0,Y 561.904,Z 611.91,A -85,B 0,C 180,E1 2839.714,E2 2839.714} C_VEL
LIN {X 0,Y 562.042,Z 611.91,A -85,B 0,C 180,E1 2845.554,E2 2845.554} C_VEL
LIN {X 0,Y 562.112,Z 611.91,A -85,B 0,C 180,E1 2851.003,E2 2851.003} C_VEL
LIN {X 0,Y 562.119,Z 611.91,A -85,B 0,C 180,E1 2856.317,E2 2856.317} C_VEL
LIN {X 0,Y 562.193,Z 611.91,A -85,B 0,C 180,E1 2861.149,E2 2861.149} C_VEL
LIN {X 0,Y 562.304,Z 611.91,A -85,B 0,C 180,E1 2867.564,E2 2867.564} C_VEL
LIN {X 0,Y 562.355,Z 611.91,A -85,B 0,C 180,E1 2872.267,E2 2872.267} C_VEL
LIN {X 0,Y 562.446,Z 611.91,A -85,B 0,C 180,E1 2876.917,E2 2876.917} C_VEL
LIN {X 0,Y 562.583,Z 611.91,A -85,B 0,C 180,E1 2881.545,E2 2881.545} C_VEL
LIN {X 0,Y 562.541,Z 611.91,A -85,B 0,C 180,E1 2886.183,E2 2886.183} C_VEL
LIN {X 0,Y 562.183,Z 611.91,A -85,B 0,C 180,E1 2892.444,E2 2892.444} C_VEL
LIN {X 0,Y 562.18,Z 611.91,A -85,B 0,C 180,E1 2897.235,E2 2897.235} C_VEL
LIN {X 0,Y 562.134,Z 611.91,A -85,B 0,C 180,E1 2902.155,E2 2902.155} C_VEL
LIN {X 0,Y 562.046,Z 611.91,A -85,B 0,C 180,E1 2907.257,E2 2907.257} C_VEL
LIN {X 0,Y 561.936,Z 611.91,A -85,B 0,C 180,E1 2912.609,E2 2912.609} C_VEL
LIN {X 0,Y 562.097,Z 611.91,A -85,B 0,C 180,E1 2918.283,E2 2918.283} C_VEL
LIN {X 0,Y 561.984,Z 611.91,A -85,B 0,C 180,E1 2924.467,E2 2924.467} C_VEL
LIN {X 0,Y 561.954,Z 611.91,A -85,B 0,C 180,E1 2929.712,E2 2929.712} C_VEL
LIN {X 0,Y 561.937,Z 611.91,A -85,B 0,C 180,E1 2935.541,E2 2935.541} C_VEL
LIN {X 0,Y 562.012,Z 611.91,A -85,B 0,C 180,E1 2940.993,E2 2940.993} C_VEL
LIN {X 0,Y 562.157,Z 611.91,A -85,B 0,C 180,E1 2946.31,E2 2946.31} C_VEL
LIN {X 0,Y 562.136,Z 611.91,A -85,B 0,C 180,E1 2951.143,E2 2951.143} C_VEL
LIN {X 0,Y 562.216,Z 611.91,A -85,B 0,C 180,E1 2955.973,E2 2955.973} C_VEL
LIN {X 0,Y 562.247,Z 611.91,A -85,B 0,C 180,E1 2960.702,E2 2960.702} C_VEL
LIN {X 0,Y 562.321,Z 611.91,A -85,B 0,C 180,E1 2965.367,E2 2965.367} C_VEL
LIN {X 0,Y 562.38,Z 611.91,A -85,B 0,C 180,E1 2970,E2 2970} C_VEL
LIN {X 0,Y 562.303,Z 611.91,A -85,B 0,C 180,E1 2974.952,E2 2974.952} C_VEL
LIN {X 0,Y 562.334,Z 611.91,A -85,B 0,C 180,E1 2979.297,E2 2979.297} C_VEL
LIN {X 0,Y 562.258,Z 611.91,A -85,B 0,C 180,E1 2984.206,E2 2984.206} C_VEL
LIN {X 0,Y 562.201,Z 611.91,A -85,B 0,C 180,E1 2989.509,E2 2989.509} C_VEL
LIN {X 0,Y 562.064,Z 611.91,A -85,B 0,C 180,E1 2995.531,E2 2995.531} C_VEL
LIN {X 0,Y 562.072,Z 611.91,A -85,B 0,C 180,E1 3000.784,E2 3000.784} C_VEL
LIN {X 0,Y 562.154,Z 611.91,A -85,B 0,C 180,E1 3006.337,E2 3006.337} C_VEL
LIN {X 0,Y 561.929,Z 611.91,A -85,B 0,C 180,E1 3012.345,E2 3012.345} C_VEL
LIN {X 0,Y 561.894,Z 611.91,A -85,B 0,C 180,E1 3017.65,E2 3017.65} C_VEL
LIN {X 0,Y 561.994,Z 611.91,A -85,B 0,C 180,E1 3023.923,E2 3023.923} C_VEL
LIN {X 0,Y 562.076,Z 611.91,A -85,B 0,C 180,E1 3029.539,E2 3029.539} C_VEL
LIN {X 0,Y 562.185,Z 611.91,A -85,B 0,C 180,E1 3034.473,E2 3034.473} C_VEL
LIN {X 0,Y 562.306,Z 611.91,A -85,B 0,C 180,E1 3040.459,E2 3040.459} C_VEL
LIN {X 0,Y 562.138,Z 611.91,A -85,B 0,C 180,E1 3044.373,E2 3044.373} C_VEL
LIN {X 0,Y 562.248,Z 611.91,A -85,B 0,C 180,E1 3050.699,E2 3050.699} C_VEL
LIN {X 0,Y 562.351,Z 611.91,A -85,B 0,C 180,E1 3055.365,E2 3055.365} C_VEL
LIN {X 0,Y 562.394,Z 611.91,A -85,B 0,C 180,E1 3059.997,E2 3059.997} C_VEL
LIN {X 0,Y 562.322,Z 611.91,A -85,B 0,C 180,E1 3064.979,E2 3064.979} C_VEL
LIN {X 0,Y 562.35,Z 611.91,A -85,B 0,C 180,E1 3069.293,E2 3069.293} C_VEL
LIN {X 0,Y 562.187,Z 611.91,A -85,B 0,C 180,E1 3074.648,E2 3074.648} C_VEL
LIN {X 0,Y 558.179,Z 611.91,A -85,B 0,C 180,E1 3076.392,E2 3076.392} C_VEL
LIN {X 0,Y 554.268,Z 611.91,A -85,B 0,C 180,E1 3078.161,E2 3078.161} C_VEL
LIN {X 0,Y 554.213,Z 611.91,A -85,B 0,C 180,E1 3084.187,E2 3084.187} C_VEL
LIN {X 0,Y 554.089,Z 611.91,A -85,B 0,C 180,E1 3089.458,E2 3089.458} C_VEL
LIN {X 0,Y 554.074,Z 611.91,A -85,B 0,C 180,E1 3095.014,E2 3095.014} C_VEL
LIN {X 0,Y 554.011,Z 611.91,A -85,B 0,C 180,E1 3100.982,E2 3100.982} C_VEL
LIN {X 0,Y 554.14,Z 611.91,A -85,B 0,C 180,E1 3106.916,E2 3106.916} C_VEL
LIN {X 0,Y 554.109,Z 611.91,A -85,B 0,C 180,E1 3113.049,E2 3113.049} C_VEL
LIN {X 0,Y 554.095,Z 611.91,A -85,B 0,C 180,E1 3118.723,E2 3118.723} C_VEL
LIN {X 0,Y 554.16,Z 612.375,A -85,B 0,C 180,E1 3121.98,E2 3121.98} C_VEL
LIN {X 0,Y 560.865,Z 629.501,A -85,B 0,C 180,E1 3122.586,E2 3122.586} C_VEL
LIN {X 0,Y 560.442,Z 673.426,A -85,B 0,C 180,E1 3123.399,E2 3123.399} C_VEL
LIN {X 0,Y 559.556,Z 711.242,A -85,B 0,C 180,E1 3124.779,E2 3124.779} C_VEL
LIN {X 0,Y 558.422,Z 744.875,A -85,B 0,C 180,E1 3126.645,E2 3126.645} C_VEL
LIN {X 0,Y 557.198,Z 776.775,A -85,B 0,C 180,E1 3129.106,E2 3129.106} C_VEL
LIN {X 0,Y 556.152,Z 805.399,A -85,B 0,C 180,E1 3132.106,E2 3132.106} C_VEL
LIN {X 0,Y 555.405,Z 829.229,A -85,B 0,C 180,E1 3135.478,E2 3135.478} C_VEL
LIN {X 0,Y 554.973,Z 847.81,A -85,B 0,C 180,E1 3139.127,E2 3139.127} C_VEL
LIN {X 0,Y 554.864,Z 860.817,A -85,B 0,C 180,E1 3142.947,E2 3142.947} C_VEL
LIN {X 0,Y 554.744,Z 868.188,A -85,B 0,C 180,E1 3146.871,E2 3146.871} C_VEL
LIN {X 0,Y 554.711,Z 870,A -85,B 0,C 180,E1 3150,E2 3150} C_VEL
LIN {X 0,Y 554.849,Z 867.168,A -85,B 0,C 180,E1 3153.912,E2 3153.912} C_VEL
LIN {X 0,Y 554.895,Z 858.629,A -85,B 0,C 180,E1 3157.841,E2 3157.841} C_VEL
LIN {X 0,Y 555.136,Z 843.704,A -85,B 0,C 180,E1 3161.803,E2 3161.803} C_VEL
LIN {X 0,Y 555.628,Z 824.032,A -85,B 0,C 180,E1 3165.346,E2 3165.346} C_VEL
LIN {X 0,Y 556.449,Z 798.81,A -85,B 0,C 180,E1 3168.671,E2 3168.671} C_VEL
LIN {X 0,Y 557.568,Z 768.483,A -85,B 0,C 180,E1 3171.61,E2 3171.61} C_VEL
LIN {X 0,Y 558.723,Z 736.354,A -85,B 0,C 180,E1 3173.891,E2 3173.891} C_VEL
LIN {X 0,Y 559.816,Z 701.678,A -85,B 0,C 180,E1 3175.641,E2 3175.641} C_VEL
LIN {X 0,Y 560.622,Z 664.094,A -85,B 0,C 180,E1 3176.83,E2 3176.83} C_VEL
LIN {X 0,Y 560.209,Z 627.855,A -85,B 0,C 180,E1 3177.472,E2 3177.472} C_VEL
LIN {X 0,Y 554.135,Z 611.91,A -85,B 0,C 180,E1 3178.121,E2 3178.121} C_VEL
LIN {X 0,Y 554.058,Z 611.91,A -85,B 0,C 180,E1 3183.129,E2 3183.129} C_VEL
LIN {X 0,Y 554.1,Z 611.91,A -85,B 0,C 180,E1 3188.937,E2 3188.937} C_VEL
LIN {X 0,Y 554.112,Z 611.91,A -85,B 0,C 180,E1 3194.737,E2 3194.737} C_VEL
LIN {X 0,Y 553.993,Z 611.91,A -85,B 0,C 180,E1 3201.06,E2 3201.06} C_VEL
LIN {X 0,Y 554.207,Z 611.91,A -85,B 0,C 180,E1 3206.885,E2 3206.885} C_VEL
LIN {X 0,Y 554.14,Z 611.91,A -85,B 0,C 180,E1 3212.328,E2 3212.328} C_VEL
LIN {X 0,Y 554.134,Z 611.91,A -85,B 0,C 180,E1 3218.276,E2 3218.276} C_VEL
LIN {X 0,Y 554.318,Z 611.91,A -85,B 0,C 180,E1 3222.937,E2 3222.937} C_VEL
LIN {X 0,Y 554.382,Z 611.91,A -85,B 0,C 180,E1 3227.383,E2 3227.383} C_VEL
LIN {X 0,Y 554.441,Z 611.91,A -85,B 0,C 180,E1 3232.156,E2 3232.156} C_VEL
LIN {X 0,Y 554.56,Z 611.91,A -85,B 0,C 180,E1 3236.873,E2 3236.873} C_VEL
LIN {X 0,Y 554.673,Z 611.91,A -85,B 0,C 180,E1 3241.567,E2 3241.567} C_VEL
LIN {X 0,Y 554.609,Z 611.91,A -85,B 0,C 180,E1 3246.272,E2 3246.272} C_VEL
LIN {X 0,Y 554.265,Z 611.91,A -85,B 0,C 180,E1 3252.625,E2 3252.625} C_VEL
LIN {X 0,Y 554.263,Z 611.91,A -85,B 0,C 180,E1 3257.489,E2 3257.489} C_VEL
LIN {X 0,Y 554.218,Z 611.91,A -85,B 0,C 180,E1 3262.488,E2 3262.488} C_VEL
LIN {X 0,Y 554.089,Z 611.91,A -85,B 0,C 180,E1 3267.682,E2 3267.682} C_VEL
LIN {X 0,Y 554.037,Z 611.91,A -85,B 0,C 180,E1 3273.133,E2 3273.133} C_VEL
LIN {X 0,Y 554.153,Z 611.91,A -85,B 0,C 180,E1 3278.934,E2 3278.934} C_VEL
LIN {X 0,Y 554.115,Z 611.91,A -85,B 0,C 180,E1 3285.271,E2 3285.271} C_VEL
LIN {X 0,Y 554.037,Z 611.91,A -85,B 0,C 180,E1 3291.058,E2 3291.058} C_VEL
LIN {X 0,Y 554.007,Z 611.91,A -85,B 0,C 180,E1 3296.867,E2 3296.867} C_VEL
LIN {X 0,Y 554.148,Z 611.91,A -85,B 0,C 180,E1 3302.324,E2 3302.324} C_VEL
LIN {X 0,Y 554.224,Z 611.91,A -85,B 0,C 180,E1 3308.255,E2 3308.255} C_VEL
LIN {X 0,Y 554.309,Z 611.91,A -85,B 0,C 180,E1 3314.149,E2 3314.149} C_VEL
LIN {X 0,Y 554.4,Z 611.91,A -85,B 0,C 180,E1 3319.471,E2 3319.471} C_VEL
LIN {X 0,Y 554.445,Z 611.91,A -85,B 0,C 180,E1 3325.301,E2 3325.301} C_VEL
LIN {X 0,Y 554.479,Z 611.91,A -85,B 0,C 180,E1 3330,E2 3330} C_VEL
LIN {X 0,Y 554.46,Z 611.91,A -85,B 0,C 180,E1 3334.699,E2 3334.699} C_VEL
LIN {X 0,Y 554.316,Z 611.91,A -85,B 0,C 180,E1 3340.482,E2 3340.482} C_VEL
LIN {X 0,Y 554.216,Z 611.91,A -85,B 0,C 180,E1 3345.854,E2 3345.854} C_VEL
LIN {X 0,Y 554.243,Z 611.91,A -85,B 0,C 180,E1 3350.801,E2 3350.801} C_VEL
LIN {X 0,Y 554.123,Z 611.91,A -85,B 0,C 180,E1 3355.924,E2 3355.924} C_VEL
LIN {X 0,Y 554.138,Z 611.91,A -85,B 0,C 180,E1 3361.274,E2 3361.274} C_VEL
LIN {X 0,Y 554.154,Z 611.91,A -85,B 0,C 180,E1 3366.947,E2 3366.947} C_VEL
LIN {X 0,Y 554.04,Z 611.91,A -85,B 0,C 180,E1 3372.45,E2 3372.45} C_VEL
LIN {X 0,Y 553.979,Z 611.91,A -85,B 0,C 180,E1 3379.008,E2 3379.008} C_VEL
LIN {X 0,Y 554.032,Z 611.91,A -85,B 0,C 180,E1 3385.068,E2 3385.068} C_VEL
LIN {X 0,Y 554.138,Z 611.91,A -85,B 0,C 180,E1 3390.965,E2 3390.965} C_VEL
LIN {X 0,Y 554.223,Z 611.91,A -85,B 0,C 180,E1 3395.807,E2 3395.807} C_VEL
LIN {X 0,Y 554.403,Z 611.91,A -85,B 0,C 180,E1 3400.868,E2 3400.868} C_VEL
LIN {X 0,Y 554.054,Z 611.91,A -85,B 0,C 180,E1 3405.76,E2 3405.76} C_VEL
LIN {X 0,Y 554.335,Z 611.91,A -85,B 0,C 180,E1 3410.565,E2 3410.565} C_VEL
LIN {X 0,Y 554.473,Z 611.91,A -85,B 0,C 180,E1 3415.298,E2 3415.298} C_VEL
LIN {X 0,Y 554.493,Z 611.91,A -85,B 0,C 180,E1 3419.997,E2 3419.997} C_VEL
LIN {X 0,Y 554.488,Z 611.91,A -85,B 0,C 180,E1 3424.696,E2 3424.696} C_VEL
LIN {X 0,Y 554.33,Z 611.91,A -85,B 0,C 180,E1 3430.493,E2 3430.493} C_VEL
LIN {X 0,Y 554.216,Z 611.91,A -85,B 0,C 180,E1 3435.85,E2 3435.85} C_VEL
LIN {X 0,Y 554.268,Z 611.91,A -85,B 0,C 180,E1 3438.161,E2 3438.161} C_VEL
LIN {X 0,Y 553.01,Z 611.91,A -85,B 0,C 180,E1 3439.054,E2 3439.054} C_VEL
LIN {X 0,Y 546.399,Z 611.91,A -85,B 0,C 180,E1 3441.484,E2 3441.484} C_VEL
LIN {X 0,Y 546.292,Z 611.91,A -85,B 0,C 180,E1 3441.714,E2 3441.714} C_VEL
LIN {X 0,Y 546.241,Z 611.91,A -85,B 0,C 180,E1 3447.506,E2 3447.506} C_VEL
LIN {X 0,Y 546.167,Z 611.91,A -85,B 0,C 180,E1 3453.732,E2 3453.732} C_VEL
LIN {X 0,Y 546.082,Z 611.91,A -85,B 0,C 180,E1 3459.614,E2 3459.614} C_VEL
LIN {X 0,Y 546.179,Z 611.91,A -85,B 0,C 180,E1 3466.13,E2 3466.13} C_VEL
LIN {X 0,Y 546.208,Z 611.91,A -85,B 0,C 180,E1 3472.423,E2 3472.423} C_VEL
LIN {X 0,Y 546.165,Z 611.91,A -85,B 0,C 180,E1 3478.217,E2 3478.217} C_VEL
LIN {X 0,Y 546.299,Z 612.624,A -85,B 0,C 180,E1 3481.544,E2 3481.544} C_VEL
LIN {X 0,Y 553.959,Z 633.966,A -85,B 0,C 180,E1 3482.279,E2 3482.279} C_VEL
LIN {X 0,Y 553.359,Z 674.584,A -85,B 0,C 180,E1 3483.064,E2 3483.064} C_VEL
LIN {X 0,Y 552.29,Z 713.204,A -85,B 0,C 180,E1 3484.515,E2 3484.515} C_VEL
LIN {X 0,Y 550.968,Z 746.998,A -85,B 0,C 180,E1 3486.46,E2 3486.46} C_VEL
LIN {X 0,Y 549.618,Z 779.064,A -85,B 0,C 180,E1 3489.015,E2 3489.015} C_VEL
LIN {X 0,Y 548.397,Z 807.34,A -85,B 0,C 180,E1 3492.086,E2 3492.086} C_VEL
LIN {X 0,Y 547.614,Z 829.872,A -85,B 0,C 180,E1 3495.375,E2 3495.375} C_VEL
LIN {X 0,Y 547.116,Z 848.544,A -85,B 0,C 180,E1 3499.139,E2 3499.139} C_VEL
LIN {X 0,Y 546.995,Z 860.812,A -85,B 0,C 180,E1 3502.845,E2 3502.845} C_VEL
LIN {X 0,Y 546.844,Z 868.191,A -85,B 0,C 180,E1 3506.826,E2 3506.826} C_VEL
LIN {X 0,Y 546.811,Z 870,A -85,B 0,C 180,E1 3510,E2 3510} C_VEL
LIN {X 0,Y 546.947,Z 867.163,A -85,B 0,C 180,E1 3513.968,E2 3513.968} C_VEL
LIN {X 0,Y 547.04,Z 858.633,A -85,B 0,C 180,E1 3517.954,E2 3517.954} C_VEL
LIN {X 0,Y 547.273,Z 843.701,A -85,B 0,C 180,E1 3521.975,E2 3521.975} C_VEL
LIN {X 0,Y 547.872,Z 823.48,A -85,B 0,C 180,E1 3525.654,E2 3525.654} C_VEL
LIN {X 0,Y 548.788,Z 799.032,A -85,B 0,C 180,E1 3528.915,E2 3528.915} C_VEL
LIN {X 0,Y 550.05,Z 768.489,A -85,B 0,C 180,E1 3531.92,E2 3531.92} C_VEL
LIN {X 0,Y 551.417,Z 736.561,A -85,B 0,C 180,E1 3534.214,E2 3534.214} C_VEL
LIN {X 0,Y 552.668,Z 701.681,A -85,B 0,C 180,E1 3535.997,E2 3535.997} C_VEL
LIN {X 0,Y 553.578,Z 664.059,A -85,B 0,C 180,E1 3537.199,E2 3537.199} C_VEL
LIN {X 0,Y 553.202,Z 630.016,A -85,B 0,C 180,E1 3537.819,E2 3537.819} C_VEL
LIN {X 0,Y 546.248,Z 611.91,A -85,B 0,C 180,E1 3538.504,E2 3538.504} C_VEL
LIN {X 0,Y 546.112,Z 611.91,A -85,B 0,C 180,E1 3543.732,E2 3543.732} C_VEL
LIN {X 0,Y 546.171,Z 611.91,A -85,B 0,C 180,E1 3549.612,E2 3549.612} C_VEL
LIN {X 0,Y 546.179,Z 611.91,A -85,B 0,C 180,E1 3553.891,E2 3553.891} C_VEL
LIN {X 0,Y 546.079,Z 611.91,A -85,B 0,C 180,E1 3560.385,E2 3560.385} C_VEL
LIN {X 0,Y 546.211,Z 611.91,A -85,B 0,C 180,E1 3566.337,E2 3566.337} C_VEL
LIN {X 0,Y 546.235,Z 611.91,A -85,B 0,C 180,E1 3571.892,E2 3571.892} C_VEL
LIN {X 0,Y 546.209,Z 611.91,A -85,B 0,C 180,E1 3577.17,E2 3577.17} C_VEL
LIN {X 0,Y 546.373,Z 611.91,A -85,B 0,C 180,E1 3582.256,E2 3582.256} C_VEL
LIN {X 0,Y 546.458,Z 611.91,A -85,B 0,C 180,E1 3587.197,E2 3587.197} C_VEL
LIN {X 0,Y 546.526,Z 611.91,A -85,B 0,C 180,E1 3592.041,E2 3592.041} C_VEL
LIN {X 0,Y 546.651,Z 611.91,A -85,B 0,C 180,E1 3596.828,E2 3596.828} C_VEL
LIN {X 0,Y 546.763,Z 611.91,A -85,B 0,C 180,E1 3601.59,E2 3601.59} C_VEL
LIN {X 0,Y 546.701,Z 611.91,A -85,B 0,C 180,E1 3606.363,E2 3606.363} C_VEL
LIN {X 0,Y 546.351,Z 611.91,A -85,B 0,C 180,E1 3612.811,E2 3612.811} C_VEL
LIN {X 0,Y 546.332,Z 611.91,A -85,B 0,C 180,E1 3617.751,E2 3617.751} C_VEL
LIN {X 0,Y 546.278,Z 611.91,A -85,B 0,C 180,E1 3622.834,E2 3622.834} C_VEL
LIN {X 0,Y 546.181,Z 611.91,A -85,B 0,C 180,E1 3628.118,E2 3628.118} C_VEL
LIN {X 0,Y 546.106,Z 611.91,A -85,B 0,C 180,E1 3633.723,E2 3633.723} C_VEL
LIN {X 0,Y 546.196,Z 611.91,A -85,B 0,C 180,E1 3639.612,E2 3639.612} C_VEL
LIN {X 0,Y 546.168,Z 611.91,A -85,B 0,C 180,E1 3646.129,E2 3646.129} C_VEL
LIN {X 0,Y 546.15,Z 611.91,A -85,B 0,C 180,E1 3652.418,E2 3652.418} C_VEL
LIN {X 0,Y 546.113,Z 611.91,A -85,B 0,C 180,E1 3658.213,E2 3658.213} C_VEL
LIN {X 0,Y 546.275,Z 611.91,A -85,B 0,C 180,E1 3663.675,E2 3663.675} C_VEL
LIN {X 0,Y 546.327,Z 611.91,A -85,B 0,C 180,E1 3668.883,E2 3668.883} C_VEL
LIN {X 0,Y 546.413,Z 611.91,A -85,B 0,C 180,E1 3673.913,E2 3673.913} C_VEL
LIN {X 0,Y 546.511,Z 611.91,A -85,B 0,C 180,E1 3678.818,E2 3678.818} C_VEL
LIN {X 0,Y 546.559,Z 611.91,A -85,B 0,C 180,E1 3685.233,E2 3685.233} C_VEL
LIN {X 0,Y 546.579,Z 611.91,A -85,B 0,C 180,E1 3690,E2 3690} C_VEL
LIN {X 0,Y 546.561,Z 611.91,A -85,B 0,C 180,E1 3694.767,E2 3694.767} C_VEL
LIN {X 0,Y 546.49,Z 611.91,A -85,B 0,C 180,E1 3699.569,E2 3699.569} C_VEL
LIN {X 0,Y 546.445,Z 611.91,A -85,B 0,C 180,E1 3704.44,E2 3704.44} C_VEL
LIN {X 0,Y 546.384,Z 611.91,A -85,B 0,C 180,E1 3709.581,E2 3709.581} C_VEL
LIN {X 0,Y 546.272,Z 611.91,A -85,B 0,C 180,E1 3714.566,E2 3714.566} C_VEL
LIN {X 0,Y 546.178,Z 611.91,A -85,B 0,C 180,E1 3719.932,E2 3719.932} C_VEL
LIN {X 0,Y 546.277,Z 611.91,A -85,B 0,C 180,E1 3725.594,E2 3725.594} C_VEL
LIN {X 0,Y 546.135,Z 611.91,A -85,B 0,C 180,E1 3731.709,E2 3731.709} C_VEL
LIN {X 0,Y 546.052,Z 611.91,A -85,B 0,C 180,E1 3738.472,E2 3738.472} C_VEL
LIN {X 0,Y 546.048,Z 611.91,A -85,B 0,C 180,E1 3744.387,E2 3744.387} C_VEL
LIN {X 0,Y 546.133,Z 611.91,A -85,B 0,C 180,E1 3750.063,E2 3750.063} C_VEL
LIN {X 0,Y 546.307,Z 611.91,A -85,B 0,C 180,E1 3756.145,E2 3756.145} C_VEL
LIN {X 0,Y 546.456,Z 611.91,A -85,B 0,C 180,E1 3760.578,E2 3760.578} C_VEL
LIN {X 0,Y 546.153,Z 611.91,A -85,B 0,C 180,E1 3765.995,E2 3765.995} C_VEL
LIN {X 0,Y 546.382,Z 611.91,A -85,B 0,C 180,E1 3771.391,E2 3771.391} C_VEL
LIN {X 0,Y 546.531,Z 611.91,A -85,B 0,C 180,E1 3775.794,E2 3775.794} C_VEL
LIN {X 0,Y 546.592,Z 611.91,A -85,B 0,C 180,E1 3779.997,E2 3779.997} C_VEL
LIN {X 0,Y 546.591,Z 611.91,A -85,B 0,C 180,E1 3784.764,E2 3784.764} C_VEL
LIN {X 0,Y 546.505,Z 611.91,A -85,B 0,C 180,E1 3789.565,E2 3789.565} C_VEL
LIN {X 0,Y 546.448,Z 611.91,A -85,B 0,C 180,E1 3794.436,E2 3794.436} C_VEL
LIN {X 0,Y 546.389,Z 611.91,A -85,B 0,C 180,E1 3799.585,E2 3799.585} C_VEL
LIN {X 0,Y 546.292,Z 611.91,A -85,B 0,C 180,E1 3801.714,E2 3801.714} C_VEL
LIN {X 0,Y 542.288,Z 611.91,A -85,B 0,C 180,E1 3803.501,E2 3803.501} C_VEL
LIN {X 0,Y 538.289,Z 611.91,A -85,B 0,C 180,E1 3805.314,E2 3805.314} C_VEL
LIN {X 0,Y 538.225,Z 611.91,A -85,B 0,C 180,E1 3810.416,E2 3810.416} C_VEL
LIN {X 0,Y 538.157,Z 611.91,A -85,B 0,C 180,E1 3816.21,E2 3816.21} C_VEL
LIN {X 0,Y 538.122,Z 611.91,A -85,B 0,C 180,E1 3822.468,E2 3822.468} C_VEL
LIN {X 0,Y 538.209,Z 611.91,A -85,B 0,C 180,E1 3827.534,E2 3827.534} C_VEL
LIN {X 0,Y 538.227,Z 611.91,A -85,B 0,C 180,E1 3833.791,E2 3833.791} C_VEL
LIN {X 0,Y 538.258,Z 611.91,A -85,B 0,C 180,E1 3839.581,E2 3839.581} C_VEL
LIN {X 0,Y 538.361,Z 611.91,A -85,B 0,C 180,E1 3841.063,E2 3841.063} C_VEL
LIN {X 0,Y 546.909,Z 633.853,A -85,B 0,C 180,E1 3841.889,E2 3841.889} C_VEL
LIN {X 0,Y 546.285,Z 675.105,A -85,B 0,C 180,E1 3842.704,E2 3842.704} C_VEL
LIN {X 0,Y 545.116,Z 712.871,A -85,B 0,C 180,E1 3844.14,E2 3844.14} C_VEL
LIN {X 0,Y 543.657,Z 746.303,A -85,B 0,C 180,E1 3846.075,E2 3846.075} C_VEL
LIN {X 0,Y 542.131,Z 777.927,A -85,B 0,C 180,E1 3848.604,E2 3848.604} C_VEL
LIN {X 0,Y 540.797,Z 805.87,A -85,B 0,C 180,E1 3851.641,E2 3851.641} C_VEL
LIN {X 0,Y 539.944,Z 828.096,A -85,B 0,C 180,E1 3854.856,E2 3854.856} C_VEL
LIN {X 0,Y 539.305,Z 847.209,A -85,B 0,C 180,E1 3858.667,E2 3858.667} C_VEL
LIN {X 0,Y 539.108,Z 859.782,A -85,B 0,C 180,E1 3862.334,E2 3862.334} C_VEL
LIN {X 0,Y 538.97,Z 867.429,A -85,B 0,C 180,E1 3866.17,E2 3866.17} C_VEL
LIN {X 0,Y 538.919,Z 870,A -85,B 0,C 180,E1 3870,E2 3870} C_VEL
LIN {X 0,Y 539.029,Z 867.357,A -85,B 0,C 180,E1 3873.882,E2 3873.882} C_VEL
LIN {X 0,Y 539.152,Z 858.636,A -85,B 0,C 180,E1 3878.072,E2 3878.072} C_VEL
LIN {X 0,Y 539.438,Z 843.698,A -85,B 0,C 180,E1 3882.152,E2 3882.152} C_VEL
LIN {X 0,Y 540.077,Z 823.62,A -85,B 0,C 180,E1 3885.863,E2 3885.863} C_VEL
LIN {X 0,Y 541.157,Z 799.035,A -85,B 0,C 180,E1 3889.193,E2 3889.193} C_VEL
LIN {X 0,Y 542.564,Z 768.492,A -85,B 0,C 180,E1 3892.239,E2 3892.239} C_VEL
LIN {X 0,Y 544.112,Z 736.722,A -85,B 0,C 180,E1 3894.55,E2 3894.55} C_VEL
LIN {X 0,Y 545.533,Z 701.684,A -85,B 0,C 180,E1 3896.363,E2 3896.363} C_VEL
LIN {X 0,Y 546.547,Z 664.044,A -85,B 0,C 180,E1 3897.578,E2 3897.578} C_VEL
LIN {X 0,Y 546.463,Z 632.763,A -85,B 0,C 180,E1 3898.152,E2 3898.152} C_VEL
LIN {X 0,Y 538.348,Z 611.91,A -85,B 0,C 180,E1 3899.023,E2 3899.023} C_VEL
LIN {X 0,Y 538.175,Z 611.91,A -85,B 0,C 180,E1 3905.336,E2 3905.336} C_VEL
LIN {X 0,Y 538.189,Z 611.91,A -85,B 0,C 180,E1 3910.581,E2 3910.581} C_VEL
LIN {X 0,Y 538.164,Z 611.91,A -85,B 0,C 180,E1 3915.311,E2 3915.311} C_VEL
LIN {X 0,Y 538.174,Z 611.91,A -85,B 0,C 180,E1 3921.974,E2 3921.974} C_VEL
LIN {X 0,Y 538.297,Z 611.91,A -85,B 0,C 180,E1 3927.701,E2 3927.701} C_VEL
LIN {X 0,Y 538.268,Z 611.91,A -85,B 0,C 180,E1 3933.257,E2 3933.257} C_VEL
LIN {X 0,Y 538.295,Z 611.91,A -85,B 0,C 180,E1 3938.557,E2 3938.557} C_VEL
LIN {X 0,Y 538.399,Z 611.91,A -85,B 0,C 180,E1 3943.671,E2 3943.671} C_VEL
LIN {X 0,Y 538.517,Z 611.91,A -85,B 0,C 180,E1 3948.653,E2 3948.653} C_VEL
LIN {X 0,Y 538.581,Z 611.91,A -85,B 0,C 180,E1 3953.547,E2 3953.547} C_VEL
LIN {X 0,Y 538.622,Z 611.91,A -85,B 0,C 180,E1 3958.392,E2 3958.392} C_VEL
LIN {X 0,Y 538.622,Z 611.91,A -85,B 0,C 180,E1 3963.226,E2 3963.226} C_VEL
LIN {X 0,Y 538.504,Z 611.91,A -85,B 0,C 180,E1 3968.084,E2 3968.084} C_VEL
LIN {X 0,Y 538.462,Z 611.91,A -85,B 0,C 180,E1 3973.002,E2 3973.002} C_VEL
LIN {X 0,Y 538.428,Z 611.91,A -85,B 0,C 180,E1 3978.021,E2 3978.021} C_VEL
LIN {X 0,Y 538.374,Z 611.91,A -85,B 0,C 180,E1 3983.188,E2 3983.188} C_VEL
LIN {X 0,Y 538.201,Z 611.91,A -85,B 0,C 180,E1 3989.298,E2 3989.298} C_VEL
LIN {X 0,Y 538.204,Z 611.91,A -85,B 0,C 180,E1 3995.332,E2 3995.332} C_VEL
LIN {X 0,Y 538.187,Z 611.91,A -85,B 0,C 180,E1 4000.573,E2 4000.573} C_VEL
LIN {X 0,Y 538.203,Z 611.91,A -85,B 0,C 180,E1 4007.008,E2 4007.008} C_VEL
LIN {X 0,Y 538.227,Z 611.91,A -85,B 0,C 180,E1 4011.968,E2 4011.968} C_VEL
LIN {X 0,Y 538.145,Z 611.91,A -85,B 0,C 180,E1 4017.686,E2 4017.686} C_VEL
LIN {X 0,Y 538.355,Z 611.91,A -85,B 0,C 180,E1 4023.258,E2 4023.258} C_VEL
LIN {X 0,Y 538.382,Z 611.91,A -85,B 0,C 180,E1 4028.556,E2 4028.556} C_VEL
LIN {X 0,Y 538.471,Z 611.91,A -85,B 0,C 180,E1 4033.67,E2 4033.67} C_VEL
LIN {X 0,Y 538.552,Z 611.91,A -85,B 0,C 180,E1 4039.731,E2 4039.731} C_VEL
LIN {X 0,Y 538.655,Z 611.91,A -85,B 0,C 180,E1 4045.163,E2 4045.163} C_VEL
LIN {X 0,Y 538.697,Z 611.91,A -85,B 0,C 180,E1 4050,E2 4050} C_VEL
LIN {X 0,Y 538.648,Z 611.91,A -85,B 0,C 180,E1 4054.837,E2 4054.837} C_VEL
LIN {X 0,Y 538.501,Z 611.91,A -85,B 0,C 180,E1 4060.239,E2 4060.239} C_VEL
LIN {X 0,Y 538.502,Z 611.91,A -85,B 0,C 180,E1 4064.658,E2 4064.658} C_VEL
LIN {X 0,Y 538.474,Z 611.91,A -85,B 0,C 180,E1 4069.719,E2 4069.719} C_VEL
LIN {X 0,Y 538.28,Z 611.91,A -85,B 0,C 180,E1 4075.829,E2 4075.829} C_VEL
LIN {X 0,Y 538.281,Z 611.91,A -85,B 0,C 180,E1 4080.417,E2 4080.417} C_VEL
LIN {X 0,Y 538.332,Z 611.91,A -85,B 0,C 180,E1 4086.201,E2 4086.201} C_VEL
LIN {X 0,Y 538.108,Z 611.91,A -85,B 0,C 180,E1 4092.476,E2 4092.476} C_VEL
LIN {X 0,Y 538.054,Z 611.91,A -85,B 0,C 180,E1 4097.517,E2 4097.517} C_VEL
LIN {X 0,Y 538.141,Z 611.91,A -85,B 0,C 180,E1 4103.782,E2 4103.782} C_VEL
LIN {X 0,Y 538.225,Z 611.91,A -85,B 0,C 180,E1 4109.577,E2 4109.577} C_VEL
LIN {X 0,Y 538.36,Z 611.91,A -85,B 0,C 180,E1 4115.046,E2 4115.046} C_VEL
LIN {X 0,Y 538.554,Z 611.91,A -85,B 0,C 180,E1 4120.282,E2 4120.282} C_VEL
LIN {X 0,Y 538.285,Z 611.91,A -85,B 0,C 180,E1 4125.334,E2 4125.334} C_VEL
LIN {X 0,Y 538.512,Z 611.91,A -85,B 0,C 180,E1 4130.286,E2 4130.286} C_VEL
LIN {X 0,Y 538.689,Z 611.91,A -85,B 0,C 180,E1 4135.16,E2 4135.16} C_VEL
LIN {X 0,Y 538.71,Z 611.91,A -85,B 0,C 180,E1 4139.997,E2 4139.997} C_VEL
LIN {X 0,Y 538.676,Z 611.91,A -85,B 0,C 180,E1 4144.834,E2 4144.834} C_VEL
LIN {X 0,Y 538.514,Z 611.91,A -85,B 0,C 180,E1 4150.251,E2 4150.251} C_VEL
LIN {X 0,Y 538.504,Z 611.91,A -85,B 0,C 180,E1 4154.654,E2 4154.654} C_VEL
LIN {X 0,Y 538.484,Z 611.91,A -85,B 0,C 180,E1 4159.715,E2 4159.715} C_VEL
LIN {X 0,Y 538.289,Z 611.91,A -85,B 0,C 180,E1 4165.314,E2 4165.314} C_VEL
LIN {X 0,Y 536.981,Z 611.91,A -85,B 0,C 180,E1 4166.237,E2 4166.237} C_VEL
LIN {X 0,Y 530.383,Z 611.91,A -85,B 0,C 180,E1 4168.75,E2 4168.75} C_VEL
LIN {X 0,Y 530.314,Z 611.91,A -85,B 0,C 180,E1 4168.988,E2 4168.988} C_VEL
LIN {X 0,Y 530.277,Z 611.91,A -85,B 0,C 180,E1 4174.818,E2 4174.818} C_VEL
LIN {X 0,Y 530.17,Z 611.91,A -85,B 0,C 180,E1 4181.053,E2 4181.053} C_VEL
LIN {X 0,Y 530.317,Z 611.91,A -85,B 0,C 180,E1 4186.749,E2 4186.749} C_VEL
LIN {X 0,Y 530.287,Z 611.91,A -85,B 0,C 180,E1 4193.069,E2 4193.069} C_VEL
LIN {X 0,Y 530.283,Z 611.91,A -85,B 0,C 180,E1 4199.074,E2 4199.074} C_VEL
LIN {X 0,Y 530.41,Z 611.91,A -85,B 0,C 180,E1 4200.589,E2 4200.589} C_VEL
LIN {X 0,Y 540.001,Z 636.359,A -85,B 0,C 180,E1 4201.533,E2 4201.533} C_VEL
LIN {X 0,Y 539.229,Z 675.59,A -85,B 0,C 180,E1 4202.334,E2 4202.334} C_VEL
LIN {X 0,Y 537.969,Z 712.488,A -85,B 0,C 180,E1 4203.753,E2 4203.753} C_VEL
LIN {X 0,Y 536.326,Z 746.288,A -85,B 0,C 180,E1 4205.726,E2 4205.726} C_VEL
LIN {X 0,Y 534.673,Z 777.974,A -85,B 0,C 180,E1 4208.295,E2 4208.295} C_VEL
LIN {X 0,Y 533.158,Z 805.862,A -85,B 0,C 180,E1 4211.369,E2 4211.369} C_VEL
LIN {X 0,Y 532.147,Z 828.742,A -85,B 0,C 180,E1 4214.741,E2 4214.741} C_VEL
LIN {X 0,Y 531.444,Z 847.207,A -85,B 0,C 180,E1 4218.497,E2 4218.497} C_VEL
LIN {X 0,Y 531.245,Z 859.784,A -85,B 0,C 180,E1 4222.22,E2 4222.22} C_VEL
LIN {X 0,Y 531.095,Z 867.416,A -85,B 0,C 180,E1 4226.107,E2 4226.107} C_VEL
LIN {X 0,Y 531.019,Z 870,A -85,B 0,C 180,E1 4230,E2 4230} C_VEL
LIN {X 0,Y 531.139,Z 867.324,A -85,B 0,C 180,E1 4233.961,E2 4233.961} C_VEL
LIN {X 0,Y 531.265,Z 858.64,A -85,B 0,C 180,E1 4238.192,E2 4238.192} C_VEL
LIN {X 0,Y 531.591,Z 843.695,A -85,B 0,C 180,E1 4242.334,E2 4242.334} C_VEL
LIN {X 0,Y 532.283,Z 824.933,A -85,B 0,C 180,E1 4245.889,E2 4245.889} C_VEL
LIN {X 0,Y 533.441,Z 800.797,A -85,B 0,C 180,E1 4249.266,E2 4249.266} C_VEL
LIN {X 0,Y 534.961,Z 771.264,A -85,B 0,C 180,E1 4252.316,E2 4252.316} C_VEL
LIN {X 0,Y 536.682,Z 739.998,A -85,B 0,C 180,E1 4254.701,E2 4254.701} C_VEL
LIN {X 0,Y 538.319,Z 703.509,A -85,B 0,C 180,E1 4256.659,E2 4256.659} C_VEL
LIN {X 0,Y 539.43,Z 667.28,A -85,B 0,C 180,E1 4257.89,E2 4257.89} C_VEL
LIN {X 0,Y 539.546,Z 634.986,A -85,B 0,C 180,E1 4258.513,E2 4258.513} C_VEL
LIN {X 0,Y 530.392,Z 611.91,A -85,B 0,C 180,E1 4259.501,E2 4259.501} C_VEL
LIN {X 0,Y 530.271,Z 611.91,A -85,B 0,C 180,E1 4264.823,E2 4264.823} C_VEL
LIN {X 0,Y 530.263,Z 611.91,A -85,B 0,C 180,E1 4271.05,E2 4271.05} C_VEL
LIN {X 0,Y 530.219,Z 611.91,A -85,B 0,C 180,E1 4276.745,E2 4276.745} C_VEL
LIN {X 0,Y 530.202,Z 611.91,A -85,B 0,C 180,E1 4283.159,E2 4283.159} C_VEL
LIN {X 0,Y 530.375,Z 611.91,A -85,B 0,C 180,E1 4289.085,E2 4289.085} C_VEL
LIN {X 0,Y 530.377,Z 611.91,A -85,B 0,C 180,E1 4294.651,E2 4294.651} C_VEL
LIN {X 0,Y 530.491,Z 611.91,A -85,B 0,C 180,E1 4300.363,E2 4300.363} C_VEL
LIN {X 0,Y 530.626,Z 611.91,A -85,B 0,C 180,E1 4306.809,E2 4306.809} C_VEL
LIN {X 0,Y 530.714,Z 611.91,A -85,B 0,C 180,E1 4311.803,E2 4311.803} C_VEL
LIN {X 0,Y 530.855,Z 611.91,A -85,B 0,C 180,E1 4316.733,E2 4316.733} C_VEL
LIN {X 0,Y 530.965,Z 611.91,A -85,B 0,C 180,E1 4321.637,E2 4321.637} C_VEL
LIN {X 0,Y 530.856,Z 611.91,A -85,B 0,C 180,E1 4326.554,E2 4326.554} C_VEL
LIN {X 0,Y 530.644,Z 611.91,A -85,B 0,C 180,E1 4331.524,E2 4331.524} C_VEL
LIN {X 0,Y 530.555,Z 611.91,A -85,B 0,C 180,E1 4336.583,E2 4336.583} C_VEL
LIN {X 0,Y 530.506,Z 611.91,A -85,B 0,C 180,E1 4341.781,E2 4341.781} C_VEL
LIN {X 0,Y 530.302,Z 611.91,A -85,B 0,C 180,E1 4347.739,E2 4347.739} C_VEL
LIN {X 0,Y 530.278,Z 611.91,A -85,B 0,C 180,E1 4354.105,E2 4354.105} C_VEL
LIN {X 0,Y 530.27,Z 611.91,A -85,B 0,C 180,E1 4359.564,E2 4359.564} C_VEL
LIN {X 0,Y 530.266,Z 611.91,A -85,B 0,C 180,E1 4365.548,E2 4365.548} C_VEL
LIN {X 0,Y 530.221,Z 611.91,A -85,B 0,C 180,E1 4371.082,E2 4371.082} C_VEL
LIN {X 0,Y 530.219,Z 611.91,A -85,B 0,C 180,E1 4377.143,E2 4377.143} C_VEL
LIN {X 0,Y 530.379,Z 611.91,A -85,B 0,C 180,E1 4382.823,E2 4382.823} C_VEL
LIN {X 0,Y 530.485,Z 611.91,A -85,B 0,C 180,E1 4388.221,E2 4388.221} C_VEL
LIN {X 0,Y 530.555,Z 611.91,A -85,B 0,C 180,E1 4393.419,E2 4393.419} C_VEL
LIN {X 0,Y 530.653,Z 611.91,A -85,B 0,C 180,E1 4398.479,E2 4398.479} C_VEL
LIN {X 0,Y 530.75,Z 611.91,A -85,B 0,C 180,E1 4405.091,E2 4405.091} C_VEL
LIN {X 0,Y 530.797,Z 611.91,A -85,B 0,C 180,E1 4410,E2 4410} C_VEL
LIN {X 0,Y 530.736,Z 611.91,A -85,B 0,C 180,E1 4414.91,E2 4414.91} C_VEL
LIN {X 0,Y 530.661,Z 611.91,A -85,B 0,C 180,E1 4419.857,E2 4419.857} C_VEL
LIN {X 0,Y 530.585,Z 611.91,A -85,B 0,C 180,E1 4424.881,E2 4424.881} C_VEL
LIN {X 0,Y 530.521,Z 611.91,A -85,B 0,C 180,E1 4430.027,E2 4430.027} C_VEL
LIN {X 0,Y 530.408,Z 611.91,A -85,B 0,C 180,E1 4435.352,E2 4435.352} C_VEL
LIN {X 0,Y 530.332,Z 611.91,A -85,B 0,C 180,E1 4441.075,E2 4441.075} C_VEL
LIN {X 0,Y 530.361,Z 611.91,A -85,B 0,C 180,E1 4446.932,E2 4446.932} C_VEL
LIN {X 0,Y 530.132,Z 611.91,A -85,B 0,C 180,E1 4453.27,E2 4453.27} C_VEL
LIN {X 0,Y 530.115,Z 611.91,A -85,B 0,C 180,E1 4458.934,E2 4458.934} C_VEL
LIN {X 0,Y 530.229,Z 611.91,A -85,B 0,C 180,E1 4465.171,E2 4465.171} C_VEL
LIN {X 0,Y 530.327,Z 611.91,A -85,B 0,C 180,E1 4470.963,E2 4470.963} C_VEL
LIN {X 0,Y 530.444,Z 611.91,A -85,B 0,C 180,E1 4476.444,E2 4476.444} C_VEL
LIN {X 0,Y 530.631,Z 611.91,A -85,B 0,C 180,E1 4481.705,E2 4481.705} C_VEL
LIN {X 0,Y 530.516,Z 611.91,A -85,B 0,C 180,E1 4488.474,E2 4488.474} C_VEL
LIN {X 0,Y 530.862,Z 611.91,A -85,B 0,C 180,E1 4493.447,E2 4493.447} C_VEL
LIN {X 0,Y 530.976,Z 611.91,A -85,B 0,C 180,E1 4498.363,E2 4498.363} C_VEL
LIN {X 0,Y 530.762,Z 611.91,A -85,B 0,C 180,E1 4504.906,E2 4504.906} C_VEL
LIN {X 0,Y 530.675,Z 611.91,A -85,B 0,C 180,E1 4509.853,E2 4509.853} C_VEL
LIN {X 0,Y 530.584,Z 611.91,A -85,B 0,C 180,E1 4514.878,E2 4514.878} C_VEL
LIN {X 0,Y 530.537,Z 611.91,A -85,B 0,C 180,E1 4520.023,E2 4520.023} C_VEL
LIN {X 0,Y 530.413,Z 611.91,A -85,B 0,C 180,E1 4525.347,E2 4525.347} C_VEL
LIN {X 0,Y 530.314,Z 611.91,A -85,B 0,C 180,E1 4528.988,E2 4528.988} C_VEL
LIN {X 0,Y 527.805,Z 611.91,A -85,B 0,C 180,E1 4530.382,E2 4530.382} C_VEL
LIN {X 0,Y 522.437,Z 611.91,A -85,B 0,C 180,E1 4532.472,E2 4532.472} C_VEL
LIN {X 0,Y 522.371,Z 611.91,A -85,B 0,C 180,E1 4532.713,E2 4532.713} C_VEL
LIN {X 0,Y 522.235,Z 611.91,A -85,B 0,C 180,E1 4538.484,E2 4538.484} C_VEL
LIN {X 0,Y 522.332,Z 611.91,A -85,B 0,C 180,E1 4544.075,E2 4544.075} C_VEL
LIN {X 0,Y 522.4,Z 611.91,A -85,B 0,C 180,E1 4550.386,E2 4550.386} C_VEL
LIN {X 0,Y 522.354,Z 611.91,A -85,B 0,C 180,E1 4556.584,E2 4556.584} C_VEL
LIN {X 0,Y 522.523,Z 612.521,A -85,B 0,C 180,E1 4560.126,E2 4560.126} C_VEL
LIN {X 0,Y 533.103,Z 639.573,A -85,B 0,C 180,E1 4561.179,E2 4561.179} C_VEL
LIN {X 0,Y 532.14,Z 678.356,A -85,B 0,C 180,E1 4562.026,E2 4562.026} C_VEL
LIN {X 0,Y 530.724,Z 715.098,A -85,B 0,C 180,E1 4563.498,E2 4563.498} C_VEL
LIN {X 0,Y 528.853,Z 749.324,A -85,B 0,C 180,E1 4565.586,E2 4565.586} C_VEL
LIN {X 0,Y 527.031,Z 780.182,A -85,B 0,C 180,E1 4568.187,E2 4568.187} C_VEL
LIN {X 0,Y 525.339,Z 809.173,A -85,B 0,C 180,E1 4571.517,E2 4571.517} C_VEL
LIN {X 0,Y 524.202,Z 832.343,A -85,B 0,C 180,E1 4575.164,E2 4575.164} C_VEL
LIN {X 0,Y 523.514,Z 849.863,A -85,B 0,C 180,E1 4578.995,E2 4578.995} C_VEL
LIN {X 0,Y 523.352,Z 860.798,A -85,B 0,C 180,E1 4582.52,E2 4582.52} C_VEL
LIN {X 0,Y 523.179,Z 868.201,A -85,B 0,C 180,E1 4586.682,E2 4586.682} C_VEL
LIN {X 0,Y 523.129,Z 870,A -85,B 0,C 180,E1 4590,E2 4590} C_VEL
LIN {X 0,Y 523.238,Z 867.319,A -85,B 0,C 180,E1 4594.021,E2 4594.021} C_VEL
LIN {X 0,Y 523.375,Z 858.643,A -85,B 0,C 180,E1 4598.317,E2 4598.317} C_VEL
LIN {X 0,Y 523.763,Z 843.692,A -85,B 0,C 180,E1 4602.521,E2 4602.521} C_VEL
LIN {X 0,Y 524.485,Z 824.929,A -85,B 0,C 180,E1 4606.132,E2 4606.132} C_VEL
LIN {X 0,Y 525.81,Z 800.801,A -85,B 0,C 180,E1 4609.557,E2 4609.557} C_VEL
LIN {X 0,Y 527.485,Z 771.794,A -85,B 0,C 180,E1 4612.599,E2 4612.599} C_VEL
LIN {X 0,Y 529.431,Z 739.999,A -85,B 0,C 180,E1 4615.062,E2 4615.062} C_VEL
LIN {X 0,Y 531.148,Z 704.686,A -85,B 0,C 180,E1 4616.99,E2 4616.99} C_VEL
LIN {X 0,Y 532.404,Z 668.984,A -85,B 0,C 180,E1 4618.246,E2 4618.246} C_VEL
LIN {X 0,Y 532.454,Z 636.885,A -85,B 0,C 180,E1 4618.9,E2 4618.9} C_VEL
LIN {X 0,Y 522.472,Z 611.91,A -85,B 0,C 180,E1 4619.916,E2 4619.916} C_VEL
LIN {X 0,Y 522.302,Z 611.91,A -85,B 0,C 180,E1 4625.749,E2 4625.749} C_VEL
LIN {X 0,Y 522.377,Z 611.91,A -85,B 0,C 180,E1 4631.808,E2 4631.808} C_VEL
LIN {X 0,Y 522.269,Z 611.91,A -85,B 0,C 180,E1 4638.188,E2 4638.188} C_VEL
LIN {X 0,Y 522.295,Z 611.91,A -85,B 0,C 180,E1 4644.571,E2 4644.571} C_VEL
LIN {X 0,Y 522.429,Z 611.91,A -85,B 0,C 180,E1 4650.488,E2 4650.488} C_VEL
LIN {X 0,Y 522.471,Z 611.91,A -85,B 0,C 180,E1 4656.069,E2 4656.069} C_VEL
LIN {X 0,Y 522.583,Z 611.91,A -85,B 0,C 180,E1 4661.42,E2 4661.42} C_VEL
LIN {X 0,Y 522.711,Z 611.91,A -85,B 0,C 180,E1 4666.605,E2 4666.605} C_VEL
LIN {X 0,Y 522.796,Z 611.91,A -85,B 0,C 180,E1 4671.677,E2 4671.677} C_VEL
LIN {X 0,Y 522.96,Z 611.91,A -85,B 0,C 180,E1 4676.684,E2 4676.684} C_VEL
LIN {X 0,Y 523.057,Z 611.91,A -85,B 0,C 180,E1 4681.662,E2 4681.662} C_VEL
LIN {X 0,Y 522.927,Z 611.91,A -85,B 0,C 180,E1 4686.653,E2 4686.653} C_VEL
LIN {X 0,Y 522.712,Z 611.91,A -85,B 0,C 180,E1 4691.701,E2 4691.701} C_VEL
LIN {X 0,Y 522.593,Z 611.91,A -85,B 0,C 180,E1 4697.045,E2 4697.045} C_VEL
LIN {X 0,Y 522.565,Z 611.91,A -85,B 0,C 180,E1 4702.129,E2 4702.129} C_VEL
LIN {X 0,Y 522.406,Z 611.91,A -85,B 0,C 180,E1 4707.629,E2 4707.629} C_VEL
LIN {X 0,Y 522.353,Z 611.91,A -85,B 0,C 180,E1 4713.419,E2 4713.419} C_VEL
LIN {X 0,Y 522.367,Z 611.91,A -85,B 0,C 180,E1 4719.619,E2 4719.619} C_VEL
LIN {X 0,Y 522.353,Z 611.91,A -85,B 0,C 180,E1 4725.921,E2 4725.921} C_VEL
LIN {X 0,Y 522.277,Z 611.91,A -85,B 0,C 180,E1 4731.512,E2 4731.512} C_VEL
LIN {X 0,Y 522.331,Z 611.91,A -85,B 0,C 180,E1 4737.206,E2 4737.206} C_VEL
LIN {X 0,Y 522.441,Z 611.91,A -85,B 0,C 180,E1 4742.375,E2 4742.375} C_VEL
LIN {X 0,Y 522.56,Z 611.91,A -85,B 0,C 180,E1 4747.999,E2 4747.999} C_VEL
LIN {X 0,Y 522.614,Z 611.91,A -85,B 0,C 180,E1 4753.16,E2 4753.16} C_VEL
LIN {X 0,Y 522.722,Z 611.91,A -85,B 0,C 180,E1 4758.302,E2 4758.302} C_VEL
LIN {X 0,Y 522.894,Z 611.91,A -85,B 0,C 180,E1 4763.349,E2 4763.349} C_VEL
LIN {X 0,Y 523.055,Z 611.91,A -85,B 0,C 180,E1 4768.341,E2 4768.341} C_VEL
LIN {X 0,Y 522.824,Z 611.91,A -85,B 0,C 180,E1 4774.984,E2 4774.984} C_VEL
LIN {X 0,Y 522.739,Z 611.91,A -85,B 0,C 180,E1 4780.008,E2 4780.008} C_VEL
LIN {X 0,Y 522.648,Z 611.91,A -85,B 0,C 180,E1 4785.113,E2 4785.113} C_VEL
LIN {X 0,Y 522.577,Z 611.91,A -85,B 0,C 180,E1 4790.345,E2 4790.345} C_VEL
LIN {X 0,Y 522.417,Z 611.91,A -85,B 0,C 180,E1 4796.045,E2 4796.045} C_VEL
LIN {X 0,Y 522.411,Z 611.91,A -85,B 0,C 180,E1 4801.445,E2 4801.445} C_VEL
LIN {X 0,Y 522.393,Z 611.91,A -85,B 0,C 180,E1 4807.491,E2 4807.491} C_VEL
LIN {X 0,Y 522.224,Z 611.91,A -85,B 0,C 180,E1 4813.545,E2 4813.545} C_VEL
LIN {X 0,Y 522.232,Z 611.91,A -85,B 0,C 180,E1 4818.92,E2 4818.92} C_VEL
LIN {X 0,Y 522.245,Z 611.91,A -85,B 0,C 180,E1 4824.56,E2 4824.56} C_VEL
LIN {X 0,Y 522.352,Z 611.91,A -85,B 0,C 180,E1 4830.476,E2 4830.476} C_VEL
LIN {X 0,Y 522.552,Z 611.91,A -85,B 0,C 180,E1 4836.067,E2 4836.067} C_VEL
LIN {X 0,Y 522.714,Z 611.91,A -85,B 0,C 180,E1 4841.418,E2 4841.418} C_VEL
LIN {X 0,Y 522.586,Z 611.91,A -85,B 0,C 180,E1 4848.296,E2 4848.296} C_VEL
LIN {X 0,Y 522.933,Z 611.91,A -85,B 0,C 180,E1 4853.347,E2 4853.347} C_VEL
LIN {X 0,Y 522.928,Z 611.91,A -85,B 0,C 180,E1 4859.997,E2 4859.997} C_VEL
LIN {X 0,Y 522.848,Z 611.91,A -85,B 0,C 180,E1 4864.981,E2 4864.981} C_VEL
LIN {X 0,Y 522.757,Z 611.91,A -85,B 0,C 180,E1 4870.023,E2 4870.023} C_VEL
LIN {X 0,Y 522.647,Z 611.91,A -85,B 0,C 180,E1 4875.109,E2 4875.109} C_VEL
LIN {X 0,Y 522.597,Z 611.91,A -85,B 0,C 180,E1 4880.34,E2 4880.34} C_VEL
LIN {X 0,Y 522.42,Z 611.91,A -85,B 0,C 180,E1 4886.048,E2 4886.048} C_VEL
LIN {X 0,Y 522.333,Z 611.91,A -85,B 0,C 180,E1 4891.445,E2 4891.445} C_VEL
LIN {X 0,Y 522.371,Z 611.91,A -85,B 0,C 180,E1 4892.713,E2 4892.713} C_VEL
LIN {X 0,Y 519.907,Z 611.91,A -85,B 0,C 180,E1 4894.125,E2 4894.125} C_VEL
LIN {X 0,Y 514.431,Z 611.91,A -85,B 0,C 180,E1 4896.241,E2 4896.241} C_VEL
LIN {X 0,Y 514.323,Z 611.91,A -85,B 0,C 180,E1 4896.486,E2 4896.486} C_VEL
LIN {X 0,Y 514.355,Z 611.91,A -85,B 0,C 180,E1 4902.617,E2 4902.617} C_VEL
LIN {X 0,Y 514.476,Z 611.91,A -85,B 0,C 180,E1 4907.401,E2 4907.401} C_VEL
LIN {X 0,Y 514.443,Z 611.91,A -85,B 0,C 180,E1 4912.613,E2 4912.613} C_VEL
LIN {X 0,Y 514.511,Z 611.91,A -85,B 0,C 180,E1 4919.367,E2 4919.367} C_VEL
LIN {X 0,Y 514.529,Z 611.91,A -85,B 0,C 180,E1 4919.598,E2 4919.598} C_VEL
LIN {X 0,Y 526.148,Z 640.649,A -85,B 0,C 180,E1 4920.781,E2 4920.781} C_VEL
LIN {X 0,Y 525.111,Z 678.586,A -85,B 0,C 180,E1 4921.63,E2 4921.63} C_VEL
LIN {X 0,Y 523.616,Z 714.561,A -85,B 0,C 180,E1 4923.08,E2 4923.08} C_VEL
LIN {X 0,Y 521.575,Z 749.319,A -85,B 0,C 180,E1 4925.222,E2 4925.222} C_VEL
LIN {X 0,Y 519.662,Z 779.065,A -85,B 0,C 180,E1 4927.743,E2 4927.743} C_VEL
LIN {X 0,Y 517.812,Z 807.521,A -85,B 0,C 180,E1 4931.017,E2 4931.017} C_VEL
LIN {X 0,Y 516.545,Z 829.924,A -85,B 0,C 180,E1 4934.487,E2 4934.487} C_VEL
LIN {X 0,Y 515.704,Z 848.429,A -85,B 0,C 180,E1 4938.441,E2 4938.441} C_VEL
LIN {X 0,Y 515.476,Z 860.793,A -85,B 0,C 180,E1 4942.405,E2 4942.405} C_VEL
LIN {X 0,Y 515.283,Z 868.204,A -85,B 0,C 180,E1 4946.631,E2 4946.631} C_VEL
LIN {X 0,Y 515.229,Z 870,A -85,B 0,C 180,E1 4950,E2 4950} C_VEL
LIN {X 0,Y 515.341,Z 867.145,A -85,B 0,C 180,E1 4954.212,E2 4954.212} C_VEL
LIN {X 0,Y 515.507,Z 858.647,A -85,B 0,C 180,E1 4958.444,E2 4958.444} C_VEL
LIN {X 0,Y 515.911,Z 843.689,A -85,B 0,C 180,E1 4962.715,E2 4962.715} C_VEL
LIN {X 0,Y 516.727,Z 824.924,A -85,B 0,C 180,E1 4966.381,E2 4966.381} C_VEL
LIN {X 0,Y 518.198,Z 800.806,A -85,B 0,C 180,E1 4969.856,E2 4969.856} C_VEL
LIN {X 0,Y 520.041,Z 771.804,A -85,B 0,C 180,E1 4972.939,E2 4972.939} C_VEL
LIN {X 0,Y 522.18,Z 739.987,A -85,B 0,C 180,E1 4975.435,E2 4975.435} C_VEL
LIN {X 0,Y 524.149,Z 703.803,A -85,B 0,C 180,E1 4977.422,E2 4977.422} C_VEL
LIN {X 0,Y 525.497,Z 667.117,A -85,B 0,C 180,E1 4978.696,E2 4978.696} C_VEL
LIN {X 0,Y 525.562,Z 639.096,A -85,B 0,C 180,E1 4979.278,E2 4979.278} C_VEL
LIN {X 0,Y 514.53,Z 611.91,A -85,B 0,C 180,E1 4980.451,E2 4980.451} C_VEL
LIN {X 0,Y 514.392,Z 611.91,A -85,B 0,C 180,E1 4986.063,E2 4986.063} C_VEL
LIN {X 0,Y 514.447,Z 611.91,A -85,B 0,C 180,E1 4990.352,E2 4990.352} C_VEL
LIN {X 0,Y 514.377,Z 611.91,A -85,B 0,C 180,E1 4995.061,E2 4995.061} C_VEL
LIN {X 0,Y 514.339,Z 611.91,A -85,B 0,C 180,E1 4999.939,E2 4999.939} C_VEL
LIN {X 0,Y 514.418,Z 611.91,A -85,B 0,C 180,E1 5006.004,E2 5006.004} C_VEL
LIN {X 0,Y 514.493,Z 611.91,A -85,B 0,C 180,E1 5011.987,E2 5011.987} C_VEL
LIN {X 0,Y 514.537,Z 611.91,A -85,B 0,C 180,E1 5017.514,E2 5017.514} C_VEL
LIN {X 0,Y 514.665,Z 611.91,A -85,B 0,C 180,E1 5022.895,E2 5022.895} C_VEL
LIN {X 0,Y 514.767,Z 611.91,A -85,B 0,C 180,E1 5028.122,E2 5028.122} C_VEL
LIN {X 0,Y 514.864,Z 611.91,A -85,B 0,C 180,E1 5033.248,E2 5033.248} C_VEL
LIN {X 0,Y 514.912,Z 611.91,A -85,B 0,C 180,E1 5038.698,E2 5038.698} C_VEL
LIN {X 0,Y 514.958,Z 611.91,A -85,B 0,C 180,E1 5043.374,E2 5043.374} C_VEL
LIN {X 0,Y 514.794,Z 611.91,A -85,B 0,C 180,E1 5048.459,E2 5048.459} C_VEL
LIN {X 0,Y 514.696,Z 611.91,A -85,B 0,C 180,E1 5053.893,E2 5053.893} C_VEL
LIN {X 0,Y 514.627,Z 611.91,A -85,B 0,C 180,E1 5059.703,E2 5059.703} C_VEL
LIN {X 0,Y 514.582,Z 611.91,A -85,B 0,C 180,E1 5064.328,E2 5064.328} C_VEL
LIN {X 0,Y 514.407,Z 611.91,A -85,B 0,C 180,E1 5070.026,E2 5070.026} C_VEL
LIN {X 0,Y 514.429,Z 611.91,A -85,B 0,C 180,E1 5076.062,E2 5076.062} C_VEL
LIN {X 0,Y 514.433,Z 611.91,A -85,B 0,C 180,E1 5080.355,E2 5080.355} C_VEL
LIN {X 0,Y 514.363,Z 611.91,A -85,B 0,C 180,E1 5085.053,E2 5085.053} C_VEL
LIN {X 0,Y 514.413,Z 611.91,A -85,B 0,C 180,E1 5089.931,E2 5089.931} C_VEL
LIN {X 0,Y 514.343,Z 611.91,A -85,B 0,C 180,E1 5095.993,E2 5095.993} C_VEL
LIN {X 0,Y 514.476,Z 611.91,A -85,B 0,C 180,E1 5101.993,E2 5101.993} C_VEL
LIN {X 0,Y 514.598,Z 611.91,A -85,B 0,C 180,E1 5107.512,E2 5107.512} C_VEL
LIN {X 0,Y 514.693,Z 611.91,A -85,B 0,C 180,E1 5112.892,E2 5112.892} C_VEL
LIN {X 0,Y 514.793,Z 611.91,A -85,B 0,C 180,E1 5118.119,E2 5118.119} C_VEL
LIN {X 0,Y 514.987,Z 611.91,A -85,B 0,C 180,E1 5123.246,E2 5123.246} C_VEL
LIN {X 0,Y 515.154,Z 611.91,A -85,B 0,C 180,E1 5128.316,E2 5128.316} C_VEL
LIN {X 0,Y 515.07,Z 611.91,A -85,B 0,C 180,E1 5133.37,E2 5133.37} C_VEL
LIN {X 0,Y 514.88,Z 611.91,A -85,B 0,C 180,E1 5138.455,E2 5138.455} C_VEL
LIN {X 0,Y 514.768,Z 611.91,A -85,B 0,C 180,E1 5143.922,E2 5143.922} C_VEL
LIN {X 0,Y 514.643,Z 611.91,A -85,B 0,C 180,E1 5149.705,E2 5149.705} C_VEL
LIN {X 0,Y 514.57,Z 611.91,A -85,B 0,C 180,E1 5154.326,E2 5154.326} C_VEL
LIN {X 0,Y 514.471,Z 611.91,A -85,B 0,C 180,E1 5160.02,E2 5160.02} C_VEL
LIN {X 0,Y 514.516,Z 611.91,A -85,B 0,C 180,E1 5166.053,E2 5166.053} C_VEL
LIN {X 0,Y 514.43,Z 611.91,A -85,B 0,C 180,E1 5170.353,E2 5170.353} C_VEL
LIN {X 0,Y 514.256,Z 611.91,A -85,B 0,C 180,E1 5177.376,E2 5177.376} C_VEL
LIN {X 0,Y 514.299,Z 611.91,A -85,B 0,C 180,E1 5182.642,E2 5182.642} C_VEL
LIN {X 0,Y 514.409,Z 611.91,A -85,B 0,C 180,E1 5188.6,E2 5188.6} C_VEL
LIN {X 0,Y 514.555,Z 611.91,A -85,B 0,C 180,E1 5193.807,E2 5193.807} C_VEL
LIN {X 0,Y 514.723,Z 611.91,A -85,B 0,C 180,E1 5200.267,E2 5200.267} C_VEL
LIN {X 0,Y 514.605,Z 611.91,A -85,B 0,C 180,E1 5204.643,E2 5204.643} C_VEL
LIN {X 0,Y 514.767,Z 611.91,A -85,B 0,C 180,E1 5209.833,E2 5209.833} C_VEL
LIN {X 0,Y 514.978,Z 611.91,A -85,B 0,C 180,E1 5214.937,E2 5214.937} C_VEL
LIN {X 0,Y 515.058,Z 611.91,A -85,B 0,C 180,E1 5219.997,E2 5219.997} C_VEL
LIN {X 0,Y 514.944,Z 611.91,A -85,B 0,C 180,E1 5225.057,E2 5225.057} C_VEL
LIN {X 0,Y 514.862,Z 611.91,A -85,B 0,C 180,E1 5230.159,E2 5230.159} C_VEL
LIN {X 0,Y 514.736,Z 611.91,A -85,B 0,C 180,E1 5235.347,E2 5235.347} C_VEL
LIN {X 0,Y 514.663,Z 611.91,A -85,B 0,C 180,E1 5240.668,E2 5240.668} C_VEL
LIN {X 0,Y 514.517,Z 611.91,A -85,B 0,C 180,E1 5246.189,E2 5246.189} C_VEL
LIN {X 0,Y 514.418,Z 611.91,A -85,B 0,C 180,E1 5251.986,E2 5251.986} C_VEL
LIN {X 0,Y 514.323,Z 611.91,A -85,B 0,C 180,E1 5256.486,E2 5256.486} C_VEL
LIN {X 0,Y 513.012,Z 611.91,A -85,B 0,C 180,E1 5257.452,E2 5257.452} C_VEL
LIN {X 0,Y 506.36,Z 611.91,A -85,B 0,C 180,E1 5260.083,E2 5260.083} C_VEL
LIN {X 0,Y 506.276,Z 611.91,A -85,B 0,C 180,E1 5260.333,E2 5260.333} C_VEL
LIN {X 0,Y 506.478,Z 611.91,A -85,B 0,C 180,E1 5266.563,E2 5266.563} C_VEL
LIN {X 0,Y 506.51,Z 611.91,A -85,B 0,C 180,E1 5273.285,E2 5273.285} C_VEL
LIN {X 0,Y 506.622,Z 612.375,A -85,B 0,C 180,E1 5279.094,E2 5279.094} C_VEL
LIN {X 0,Y 519.16,Z 642.609,A -85,B 0,C 180,E1 5280.383,E2 5280.383} C_VEL
LIN {X 0,Y 517.983,Z 682.828,A -85,B 0,C 180,E1 5281.357,E2 5281.357} C_VEL
LIN {X 0,Y 516.232,Z 718.498,A -85,B 0,C 180,E1 5282.902,E2 5282.902} C_VEL
LIN {X 0,Y 513.98,Z 753.873,A -85,B 0,C 180,E1 5285.18,E2 5285.18} C_VEL
LIN {X 0,Y 511.731,Z 785.267,A -85,B 0,C 180,E1 5288.052,E2 5288.052} C_VEL
LIN {X 0,Y 509.924,Z 811.229,A -85,B 0,C 180,E1 5291.232,E2 5291.232} C_VEL
LIN {X 0,Y 508.528,Z 834.784,A -85,B 0,C 180,E1 5295.162,E2 5295.162} C_VEL
LIN {X 0,Y 507.746,Z 851.974,A -85,B 0,C 180,E1 5299.259,E2 5299.259} C_VEL
LIN {X 0,Y 507.509,Z 862.784,A -85,B 0,C 180,E1 5303.146,E2 5303.146} C_VEL
LIN {X 0,Y 507.382,Z 868.207,A -85,B 0,C 180,E1 5306.579,E2 5306.579} C_VEL
LIN {X 0,Y 507.342,Z 870,A -85,B 0,C 180,E1 5310,E2 5310} C_VEL
LIN {X 0,Y 507.44,Z 867.141,A -85,B 0,C 180,E1 5314.278,E2 5314.278} C_VEL
LIN {X 0,Y 507.612,Z 858.649,A -85,B 0,C 180,E1 5318.577,E2 5318.577} C_VEL
LIN {X 0,Y 508.078,Z 843.687,A -85,B 0,C 180,E1 5322.915,E2 5322.915} C_VEL
LIN {X 0,Y 508.996,Z 824.919,A -85,B 0,C 180,E1 5326.637,E2 5326.637} C_VEL
LIN {X 0,Y 510.617,Z 800.809,A -85,B 0,C 180,E1 5330.163,E2 5330.163} C_VEL
LIN {X 0,Y 512.688,Z 771.248,A -85,B 0,C 180,E1 5333.34,E2 5333.34} C_VEL
LIN {X 0,Y 514.956,Z 739.912,A -85,B 0,C 180,E1 5335.818,E2 5335.818} C_VEL
LIN {X 0,Y 517.055,Z 703.792,A -85,B 0,C 180,E1 5337.819,E2 5337.819} C_VEL
LIN {X 0,Y 518.507,Z 668.592,A -85,B 0,C 180,E1 5339.074,E2 5339.074} C_VEL
LIN {X 0,Y 518.804,Z 641.7,A -85,B 0,C 180,E1 5339.653,E2 5339.653} C_VEL
LIN {X 0,Y 506.584,Z 611.91,A -85,B 0,C 180,E1 5340.998,E2 5340.998} C_VEL
LIN {X 0,Y 506.491,Z 611.91,A -85,B 0,C 180,E1 5346.717,E2 5346.717} C_VEL
LIN {X 0,Y 506.455,Z 611.91,A -85,B 0,C 180,E1 5353.44,E2 5353.44} C_VEL
LIN {X 0,Y 506.353,Z 611.91,A -85,B 0,C 180,E1 5358.872,E2 5358.872} C_VEL
LIN {X 0,Y 506.485,Z 611.91,A -85,B 0,C 180,E1 5365.396,E2 5365.396} C_VEL
LIN {X 0,Y 506.536,Z 611.91,A -85,B 0,C 180,E1 5371.434,E2 5371.434} C_VEL
LIN {X 0,Y 506.626,Z 611.91,A -85,B 0,C 180,E1 5377.886,E2 5377.886} C_VEL
LIN {X 0,Y 506.772,Z 611.91,A -85,B 0,C 180,E1 5382.949,E2 5382.949} C_VEL
LIN {X 0,Y 506.846,Z 611.91,A -85,B 0,C 180,E1 5387.934,E2 5387.934} C_VEL
LIN {X 0,Y 506.954,Z 611.91,A -85,B 0,C 180,E1 5393.142,E2 5393.142} C_VEL
LIN {X 0,Y 507.059,Z 611.91,A -85,B 0,C 180,E1 5398.292,E2 5398.292} C_VEL
LIN {X 0,Y 507.053,Z 611.91,A -85,B 0,C 180,E1 5403.427,E2 5403.427} C_VEL
LIN {X 0,Y 506.88,Z 611.91,A -85,B 0,C 180,E1 5408.592,E2 5408.592} C_VEL
LIN {X 0,Y 506.809,Z 611.91,A -85,B 0,C 180,E1 5413.83,E2 5413.83} C_VEL
LIN {X 0,Y 506.728,Z 611.91,A -85,B 0,C 180,E1 5419.191,E2 5419.191} C_VEL
LIN {X 0,Y 506.625,Z 611.91,A -85,B 0,C 180,E1 5424.735,E2 5424.735} C_VEL
LIN {X 0,Y 506.488,Z 611.91,A -85,B 0,C 180,E1 5430.545,E2 5430.545} C_VEL
LIN {X 0,Y 506.532,Z 611.91,A -85,B 0,C 180,E1 5436.715,E2 5436.715} C_VEL
LIN {X 0,Y 506.394,Z 611.91,A -85,B 0,C 180,E1 5443.448,E2 5443.448} C_VEL
LIN {X 0,Y 506.423,Z 611.91,A -85,B 0,C 180,E1 5448.873,E2 5448.873} C_VEL
LIN {X 0,Y 506.431,Z 611.91,A -85,B 0,C 180,E1 5455.387,E2 5455.387} C_VEL
LIN {X 0,Y 506.497,Z 611.91,A -85,B 0,C 180,E1 5461.427,E2 5461.427} C_VEL
LIN {X 0,Y 506.69,Z 611.91,A -85,B 0,C 180,E1 5467.141,E2 5467.141} C_VEL
LIN {X 0,Y 506.787,Z 611.91,A -85,B 0,C 180,E1 5472.947,E2 5472.947} C_VEL
LIN {X 0,Y 506.864,Z 611.91,A -85,B 0,C 180,E1 5477.931,E2 5477.931} C_VEL
LIN {X 0,Y 507.059,Z 611.91,A -85,B 0,C 180,E1 5483.14,E2 5483.14} C_VEL
LIN {X 0,Y 507.271,Z 611.91,A -85,B 0,C 180,E1 5488.29,E2 5488.29} C_VEL
LIN {X 0,Y 507.158,Z 611.91,A -85,B 0,C 180,E1 5493.423,E2 5493.423} C_VEL
LIN {X 0,Y 506.897,Z 611.91,A -85,B 0,C 180,E1 5499.704,E2 5499.704} C_VEL
LIN {X 0,Y 506.802,Z 611.91,A -85,B 0,C 180,E1 5505.597,E2 5505.597} C_VEL
LIN {X 0,Y 506.689,Z 611.91,A -85,B 0,C 180,E1 5511.013,E2 5511.013} C_VEL
LIN {X 0,Y 506.583,Z 611.91,A -85,B 0,C 180,E1 5516.636,E2 5516.636} C_VEL
LIN {X 0,Y 506.564,Z 611.91,A -85,B 0,C 180,E1 5522.547,E2 5522.547} C_VEL
LIN {X 0,Y 506.587,Z 611.91,A -85,B 0,C 180,E1 5526.709,E2 5526.709} C_VEL
LIN {X 0,Y 506.363,Z 611.91,A -85,B 0,C 180,E1 5531.622,E2 5531.622} C_VEL
LIN {X 0,Y 506.271,Z 611.91,A -85,B 0,C 180,E1 5538.387,E2 5538.387} C_VEL
LIN {X 0,Y 506.419,Z 611.91,A -85,B 0,C 180,E1 5543.826,E2 5543.826} C_VEL
LIN {X 0,Y 506.514,Z 611.91,A -85,B 0,C 180,E1 5550.095,E2 5550.095} C_VEL
LIN {X 0,Y 506.652,Z 611.91,A -85,B 0,C 180,E1 5555.266,E2 5555.266} C_VEL
LIN {X 0,Y 506.854,Z 611.91,A -85,B 0,C 180,E1 5560.814,E2 5560.814} C_VEL
LIN {X 0,Y 506.632,Z 611.91,A -85,B 0,C 180,E1 5566.165,E2 5566.165} C_VEL
LIN {X 0,Y 506.877,Z 611.91,A -85,B 0,C 180,E1 5571.425,E2 5571.425} C_VEL
LIN {X 0,Y 507.053,Z 611.91,A -85,B 0,C 180,E1 5576.573,E2 5576.573} C_VEL
LIN {X 0,Y 507.059,Z 611.91,A -85,B 0,C 180,E1 5581.708,E2 5581.708} C_VEL
LIN {X 0,Y 506.946,Z 611.91,A -85,B 0,C 180,E1 5586.858,E2 5586.858} C_VEL
LIN {X 0,Y 506.848,Z 611.91,A -85,B 0,C 180,E1 5592.066,E2 5592.066} C_VEL
LIN {X 0,Y 506.773,Z 611.91,A -85,B 0,C 180,E1 5597.379,E2 5597.379} C_VEL
LIN {X 0,Y 506.703,Z 611.91,A -85,B 0,C 180,E1 5602.854,E2 5602.854} C_VEL
LIN {X 0,Y 506.482,Z 611.91,A -85,B 0,C 180,E1 5608.569,E2 5608.569} C_VEL
LIN {X 0,Y 506.461,Z 611.91,A -85,B 0,C 180,E1 5614.606,E2 5614.606} C_VEL
